LIN {X 0,Y 156.666,Z 359.376,A -85,B 0,C 180,E1 -23638.457,E2 -23638.457} C_VEL
LIN {X 0,Y 158.288,Z 353.415,A -85,B 0,C 180,E1 -23642.612,E2 -23642.612} C_VEL
LIN {X 0,Y 160.591,Z 345.69,A -85,B 0,C 180,E1 -23646.772,E2 -23646.772} C_VEL
LIN {X 0,Y 163.163,Z 336.899,A -85,B 0,C 180,E1 -23650.436,E2 -23650.436} C_VEL
LIN {X 0,Y 166.03,Z 327.188,A -85,B 0,C 180,E1 -23653.61,E2 -23653.61} C_VEL
LIN {X 0,Y 168.599,Z 317.53,A -85,B 0,C 180,E1 -23656.133,E2 -23656.133} C_VEL
LIN {X 0,Y 169.428,Z 313.24,A -85,B 0,C 180,E1 -23657.118,E2 -23657.118} C_VEL
LIN {X 0,Y 167.813,Z 301.872,A -85,B 0,C 180,E1 -23659.907,E2 -23659.907} C_VEL
LIN {X 0,Y 165.385,Z 290.388,A -85,B 0,C 180,E1 -23662.401,E2 -23662.401} C_VEL
LIN {X 0,Y 162.961,Z 281.712,A -85,B 0,C 180,E1 -23664.133,E2 -23664.133} C_VEL
LIN {X 0,Y 157.967,Z 269.688,A -85,B 0,C 180,E1 -23666.494,E2 -23666.494} C_VEL
LIN {X 0,Y 157.834,Z 268.828,A -85,B 0,C 180,E1 -23666.651,E2 -23666.651} C_VEL
LIN {X 0,Y 158.243,Z 268.777,A -85,B 0,C 180,E1 -23670.001,E2 -23670.001} C_VEL
LIN {X 0,Y 157.797,Z 268.827,A -85,B 0,C 180,E1 -23677.68,E2 -23677.68} C_VEL
LIN {X 0,Y 157.671,Z 268.84,A -85,B 0,C 180,E1 -23681.324,E2 -23681.324} C_VEL
LIN {X 0,Y 157.478,Z 268.873,A -85,B 0,C 180,E1 -23685.533,E2 -23685.533} C_VEL
LIN {X 0,Y 157.406,Z 268.881,A -85,B 0,C 180,E1 -23690.929,E2 -23690.929} C_VEL
LIN {X 0,Y 157.309,Z 268.883,A -85,B 0,C 180,E1 -23696.691,E2 -23696.691} C_VEL
LIN {X 0,Y 157.275,Z 268.897,A -85,B 0,C 180,E1 -23702.429,E2 -23702.429} C_VEL
LIN {X 0,Y 157.317,Z 268.876,A -85,B 0,C 180,E1 -23706.482,E2 -23706.482} C_VEL
LIN {X 0,Y 157.29,Z 268.893,A -85,B 0,C 180,E1 -23712.086,E2 -23712.086} C_VEL
LIN {X 0,Y 157.307,Z 268.881,A -85,B 0,C 180,E1 -23715.631,E2 -23715.631} C_VEL
LIN {X 0,Y 157.29,Z 268.889,A -85,B 0,C 180,E1 -23721.284,E2 -23721.284} C_VEL
LIN {X 0,Y 157.309,Z 268.889,A -85,B 0,C 180,E1 -23724.5,E2 -23724.5} C_VEL
LIN {X 0,Y 157.292,Z 268.878,A -85,B 0,C 180,E1 -23728.099,E2 -23728.099} C_VEL
LIN {X 0,Y 157.32,Z 268.883,A -85,B 0,C 180,E1 -23733.471,E2 -23733.471} C_VEL
LIN {X 0,Y 157.394,Z 268.872,A -85,B 0,C 180,E1 -23739.672,E2 -23739.672} C_VEL
LIN {X 0,Y 157.454,Z 268.858,A -85,B 0,C 180,E1 -23744.471,E2 -23744.471} C_VEL
LIN {X 0,Y 157.691,Z 268.843,A -85,B 0,C 180,E1 -23749.735,E2 -23749.735} C_VEL
LIN {X 0,Y 157.768,Z 268.826,A -85,B 0,C 180,E1 -23752.324,E2 -23752.324} C_VEL
LIN {X 0,Y 158.26,Z 268.771,A -85,B 0,C 180,E1 -23760.004,E2 -23760.004} C_VEL
LIN {X 0,Y 157.768,Z 268.819,A -85,B 0,C 180,E1 -23767.684,E2 -23767.684} C_VEL
LIN {X 0,Y 157.643,Z 268.848,A -85,B 0,C 180,E1 -23771.24,E2 -23771.24} C_VEL
LIN {X 0,Y 157.46,Z 268.861,A -85,B 0,C 180,E1 -23775.538,E2 -23775.538} C_VEL
LIN {X 0,Y 157.378,Z 268.881,A -85,B 0,C 180,E1 -23780.936,E2 -23780.936} C_VEL
LIN {X 0,Y 157.323,Z 268.889,A -85,B 0,C 180,E1 -23786.687,E2 -23786.687} C_VEL
LIN {X 0,Y 157.376,Z 269.021,A -85,B 0,C 180,E1 -23790.534,E2 -23790.534} C_VEL
LIN {X 0,Y 158.013,Z 272.957,A -85,B 0,C 180,E1 -23796.811,E2 -23796.811} C_VEL
LIN {X 0,Y 158.647,Z 276.209,A -85,B 0,C 180,E1 -23801.648,E2 -23801.648} C_VEL
LIN {X 0,Y 159.409,Z 279.832,A -85,B 0,C 180,E1 -23806.677,E2 -23806.677} C_VEL
LIN {X 0,Y 159.866,Z 282.353,A -85,B 0,C 180,E1 -23810.02,E2 -23810.02} C_VEL
LIN {X 0,Y 160.877,Z 285.754,A -85,B 0,C 180,E1 -23810.495,E2 -23810.495} C_VEL
LIN {X 0,Y 162.697,Z 294.146,A -85,B 0,C 180,E1 -23811.682,E2 -23811.682} C_VEL
LIN {X 0,Y 164.39,Z 306.903,A -85,B 0,C 180,E1 -23813.661,E2 -23813.661} C_VEL
LIN {X 0,Y 165.271,Z 319.319,A -85,B 0,C 180,E1 -23815.96,E2 -23815.96} C_VEL
LIN {X 0,Y 165.657,Z 331.535,A -85,B 0,C 180,E1 -23818.672,E2 -23818.672} C_VEL
LIN {X 0,Y 165.429,Z 342.008,A -85,B 0,C 180,E1 -23821.448,E2 -23821.448} C_VEL
LIN {X 0,Y 164.94,Z 346.369,A -85,B 0,C 180,E1 -23822.737,E2 -23822.737} C_VEL
LIN {X 0,Y 161.879,Z 356.685,A -85,B 0,C 180,E1 -23826.202,E2 -23826.202} C_VEL
LIN {X 0,Y 159.671,Z 364.153,A -85,B 0,C 180,E1 -23829.381,E2 -23829.381} C_VEL
LIN {X 0,Y 157.6,Z 371.203,A -85,B 0,C 180,E1 -23833.149,E2 -23833.149} C_VEL
LIN {X 0,Y 156.217,Z 376.821,A -85,B 0,C 180,E1 -23836.999,E2 -23836.999} C_VEL
LIN {X 0,Y 155.439,Z 381.221,A -85,B 0,C 180,E1 -23840.893,E2 -23840.893} C_VEL
LIN {X 0,Y 155.223,Z 384.632,A -85,B 0,C 180,E1 -23844.97,E2 -23844.97} C_VEL
LIN {X 0,Y 155.246,Z 386.125,A -85,B 0,C 180,E1 -23847.404,E2 -23847.404} C_VEL
LIN {X 0,Y 155.289,Z 387.302,A -85,B 0,C 180,E1 -23849.999,E2 -23849.999} C_VEL
LIN {X 0,Y 155.064,Z 388.289,A -85,B 0,C 180,E1 -23854.31,E2 -23854.31} C_VEL
LIN {X 0,Y 155.115,Z 388.283,A -85,B 0,C 180,E1 -23857.811,E2 -23857.811} C_VEL
LIN {X 0,Y 156.078,Z 387.02,A -85,B 0,C 180,E1 -23863.01,E2 -23863.01} C_VEL
LIN {X 0,Y 156.979,Z 385.836,A -85,B 0,C 180,E1 -23865.581,E2 -23865.581} C_VEL
LIN {X 0,Y 159.942,Z 382.247,A -85,B 0,C 180,E1 -23870.579,E2 -23870.579} C_VEL
LIN {X 0,Y 162.874,Z 378.482,A -85,B 0,C 180,E1 -23874.198,E2 -23874.198} C_VEL
LIN {X 0,Y 166.42,Z 373.702,A -85,B 0,C 180,E1 -23877.678,E2 -23877.678} C_VEL
LIN {X 0,Y 171.352,Z 366.713,A -85,B 0,C 180,E1 -23881.528,E2 -23881.528} C_VEL
LIN {X 0,Y 176.356,Z 359.27,A -85,B 0,C 180,E1 -23884.601,E2 -23884.601} C_VEL
LIN {X 0,Y 179.653,Z 351.998,A -85,B 0,C 180,E1 -23887.325,E2 -23887.325} C_VEL
LIN {X 0,Y 181.699,Z 345.766,A -85,B 0,C 180,E1 -23889.535,E2 -23889.535} C_VEL
LIN {X 0,Y 182.216,Z 342.101,A -85,B 0,C 180,E1 -23890.981,E2 -23890.981} C_VEL
LIN {X 0,Y 181.948,Z 338.759,A -85,B 0,C 180,E1 -23892.537,E2 -23892.537} C_VEL
LIN {X 0,Y 179.479,Z 328.783,A -85,B 0,C 180,E1 -23898.053,E2 -23898.053} C_VEL
LIN {X 0,Y 178.576,Z 323.642,A -85,B 0,C 180,E1 -23900.969,E2 -23900.969} C_VEL
LIN {X 0,Y 177.655,Z 319.569,A -85,B 0,C 180,E1 -23903.597,E2 -23903.597} C_VEL
LIN {X 0,Y 176.426,Z 314.669,A -85,B 0,C 180,E1 -23907.462,E2 -23907.462} C_VEL
LIN {X 0,Y 175.05,Z 309.179,A -85,B 0,C 180,E1 -23913.788,E2 -23913.788} C_VEL
LIN {X 0,Y 174.616,Z 307.537,A -85,B 0,C 180,E1 -23917.771,E2 -23917.771} C_VEL
LIN {X 0,Y 174.771,Z 306.887,A -85,B 0,C 180,E1 -23921.23,E2 -23921.23} C_VEL
LIN {X 0,Y 175.305,Z 306.933,A -85,B 0,C 180,E1 -23924.183,E2 -23924.183} C_VEL
LIN {X 0,Y 177.03,Z 310.07,A -85,B 0,C 180,E1 -23930.859,E2 -23930.859} C_VEL
LIN {X 0,Y 178.903,Z 314.102,A -85,B 0,C 180,E1 -23935.49,E2 -23935.49} C_VEL
LIN {X 0,Y 180.062,Z 318.511,A -85,B 0,C 180,E1 -23938.878,E2 -23938.878} C_VEL
LIN {X 0,Y 181.071,Z 323.62,A -85,B 0,C 180,E1 -23942.221,E2 -23942.221} C_VEL
LIN {X 0,Y 181.258,Z 328.749,A -85,B 0,C 180,E1 -23945.001,E2 -23945.001} C_VEL
LIN {X 0,Y 180.673,Z 334.595,A -85,B 0,C 180,E1 -23947.821,E2 -23947.821} C_VEL
LIN {X 0,Y 179.865,Z 337.31,A -85,B 0,C 180,E1 -23948.988,E2 -23948.988} C_VEL
LIN {X 0,Y 174.797,Z 345.135,A -85,B 0,C 180,E1 -23951.593,E2 -23951.593} C_VEL
LIN {X 0,Y 169.011,Z 352.991,A -85,B 0,C 180,E1 -23955.049,E2 -23955.049} C_VEL
LIN {X 0,Y 163.515,Z 359.573,A -85,B 0,C 180,E1 -23958.994,E2 -23958.994} C_VEL
LIN {X 0,Y 159.609,Z 363.69,A -85,B 0,C 180,E1 -23962.384,E2 -23962.384} C_VEL
LIN {X 0,Y 155.548,Z 367.521,A -85,B 0,C 180,E1 -23966.855,E2 -23966.855} C_VEL
LIN {X 0,Y 153.024,Z 369.486,A -85,B 0,C 180,E1 -23970.339,E2 -23970.339} C_VEL
LIN {X 0,Y 150.989,Z 370.683,A -85,B 0,C 180,E1 -23973.95,E2 -23973.95} C_VEL
LIN {X 0,Y 149.468,Z 371.159,A -85,B 0,C 180,E1 -23977.674,E2 -23977.674} C_VEL
LIN {X 0,Y 148.38,Z 370.887,A -85,B 0,C 180,E1 -23981.53,E2 -23981.53} C_VEL
LIN {X 0,Y 147.801,Z 369.765,A -85,B 0,C 180,E1 -23985.493,E2 -23985.493} C_VEL
LIN {X 0,Y 147.748,Z 367.741,A -85,B 0,C 180,E1 -23989.552,E2 -23989.552} C_VEL
LIN {X 0,Y 148.32,Z 364.749,A -85,B 0,C 180,E1 -23993.652,E2 -23993.652} C_VEL
LIN {X 0,Y 149.366,Z 360.568,A -85,B 0,C 180,E1 -23997.87,E2 -23997.87} C_VEL
LIN {X 0,Y 150.925,Z 354.855,A -85,B 0,C 180,E1 -24002.249,E2 -24002.249} C_VEL
LIN {X 0,Y 153.216,Z 347.505,A -85,B 0,C 180,E1 -24006.535,E2 -24006.535} C_VEL
LIN {X 0,Y 155.853,Z 338.829,A -85,B 0,C 180,E1 -24010.487,E2 -24010.487} C_VEL
LIN {X 0,Y 158.843,Z 328.979,A -85,B 0,C 180,E1 -24013.948,E2 -24013.948} C_VEL
LIN {X 0,Y 161.788,Z 318.591,A -85,B 0,C 180,E1 -24016.819,E2 -24016.819} C_VEL
LIN {X 0,Y 162.665,Z 314.349,A -85,B 0,C 180,E1 -24017.842,E2 -24017.842} C_VEL
LIN {X 0,Y 161.407,Z 304.628,A -85,B 0,C 180,E1 -24020.395,E2 -24020.395} C_VEL
LIN {X 0,Y 159.163,Z 293.185,A -85,B 0,C 180,E1 -24023.068,E2 -24023.068} C_VEL
LIN {X 0,Y 156.904,Z 284.815,A -85,B 0,C 180,E1 -24024.862,E2 -24024.862} C_VEL
LIN {X 0,Y 151.838,Z 272.437,A -85,B 0,C 180,E1 -24027.556,E2 -24027.556} C_VEL
LIN {X 0,Y 150.939,Z 269.688,A -85,B 0,C 180,E1 -24028.084,E2 -24028.084} C_VEL
LIN {X 0,Y 151.203,Z 269.654,A -85,B 0,C 180,E1 -24030.001,E2 -24030.001} C_VEL
LIN {X 0,Y 150.732,Z 269.709,A -85,B 0,C 180,E1 -24038.042,E2 -24038.042} C_VEL
LIN {X 0,Y 150.602,Z 269.72,A -85,B 0,C 180,E1 -24041.51,E2 -24041.51} C_VEL
LIN {X 0,Y 150.387,Z 269.757,A -85,B 0,C 180,E1 -24046.285,E2 -24046.285} C_VEL
LIN {X 0,Y 150.379,Z 269.756,A -85,B 0,C 180,E1 -24050.835,E2 -24050.835} C_VEL
LIN {X 0,Y 150.238,Z 269.763,A -85,B 0,C 180,E1 -24057.288,E2 -24057.288} C_VEL
LIN {X 0,Y 150.215,Z 269.775,A -85,B 0,C 180,E1 -24062.641,E2 -24062.641} C_VEL
LIN {X 0,Y 150.229,Z 269.761,A -85,B 0,C 180,E1 -24067.459,E2 -24067.459} C_VEL
LIN {X 0,Y 150.231,Z 269.771,A -85,B 0,C 180,E1 -24071.547,E2 -24071.547} C_VEL
LIN {X 0,Y 150.282,Z 269.756,A -85,B 0,C 180,E1 -24075.461,E2 -24075.461} C_VEL
LIN {X 0,Y 150.232,Z 269.759,A -85,B 0,C 180,E1 -24079.092,E2 -24079.092} C_VEL
LIN {X 0,Y 150.268,Z 269.767,A -85,B 0,C 180,E1 -24082.665,E2 -24082.665} C_VEL
LIN {X 0,Y 150.218,Z 269.764,A -85,B 0,C 180,E1 -24087.369,E2 -24087.369} C_VEL
LIN {X 0,Y 150.242,Z 269.762,A -85,B 0,C 180,E1 -24092.723,E2 -24092.723} C_VEL
LIN {X 0,Y 150.35,Z 269.751,A -85,B 0,C 180,E1 -24099.213,E2 -24099.213} C_VEL
LIN {X 0,Y 150.361,Z 269.736,A -85,B 0,C 180,E1 -24103.718,E2 -24103.718} C_VEL
LIN {X 0,Y 150.613,Z 269.723,A -85,B 0,C 180,E1 -24109.247,E2 -24109.247} C_VEL
LIN {X 0,Y 150.706,Z 269.707,A -85,B 0,C 180,E1 -24111.962,E2 -24111.962} C_VEL
LIN {X 0,Y 151.221,Z 269.648,A -85,B 0,C 180,E1 -24120.004,E2 -24120.004} C_VEL
LIN {X 0,Y 150.706,Z 269.701,A -85,B 0,C 180,E1 -24128.047,E2 -24128.047} C_VEL
LIN {X 0,Y 150.583,Z 269.728,A -85,B 0,C 180,E1 -24131.44,E2 -24131.44} C_VEL
LIN {X 0,Y 150.367,Z 269.743,A -85,B 0,C 180,E1 -24136.29,E2 -24136.29} C_VEL
LIN {X 0,Y 150.359,Z 269.755,A -85,B 0,C 180,E1 -24140.796,E2 -24140.796} C_VEL
LIN {X 0,Y 150.254,Z 269.769,A -85,B 0,C 180,E1 -24147.286,E2 -24147.286} C_VEL
LIN {X 0,Y 150.284,Z 269.815,A -85,B 0,C 180,E1 -24149.798,E2 -24149.798} C_VEL
LIN {X 0,Y 150.664,Z 272.327,A -85,B 0,C 180,E1 -24154.044,E2 -24154.044} C_VEL
LIN {X 0,Y 151.126,Z 274.608,A -85,B 0,C 180,E1 -24157.759,E2 -24157.759} C_VEL
LIN {X 0,Y 151.921,Z 278.719,A -85,B 0,C 180,E1 -24163.946,E2 -24163.946} C_VEL
LIN {X 0,Y 152.638,Z 282.108,A -85,B 0,C 180,E1 -24168.532,E2 -24168.532} C_VEL
LIN {X 0,Y 153.768,Z 285.468,A -85,B 0,C 180,E1 -24169.066,E2 -24169.066} C_VEL
LIN {X 0,Y 155.923,Z 293.086,A -85,B 0,C 180,E1 -24170.301,E2 -24170.301} C_VEL
LIN {X 0,Y 157.671,Z 305.728,A -85,B 0,C 180,E1 -24172.338,E2 -24172.338} C_VEL
LIN {X 0,Y 158.46,Z 316.907,A -85,B 0,C 180,E1 -24174.449,E2 -24174.449} C_VEL
LIN {X 0,Y 158.758,Z 329.337,A -85,B 0,C 180,E1 -24177.263,E2 -24177.263} C_VEL
LIN {X 0,Y 158.629,Z 339.851,A -85,B 0,C 180,E1 -24180.103,E2 -24180.103} C_VEL
LIN {X 0,Y 158.315,Z 345.557,A -85,B 0,C 180,E1 -24181.856,E2 -24181.856} C_VEL
LIN {X 0,Y 155.24,Z 355.549,A -85,B 0,C 180,E1 -24185.303,E2 -24185.303} C_VEL
LIN {X 0,Y 152.604,Z 364.128,A -85,B 0,C 180,E1 -24189.088,E2 -24189.088} C_VEL
LIN {X 0,Y 150.499,Z 371.077,A -85,B 0,C 180,E1 -24193.029,E2 -24193.029} C_VEL
LIN {X 0,Y 148.93,Z 377.433,A -85,B 0,C 180,E1 -24197.738,E2 -24197.738} C_VEL
LIN {X 0,Y 148.275,Z 381.585,A -85,B 0,C 180,E1 -24201.824,E2 -24201.824} C_VEL
LIN {X 0,Y 148.144,Z 384.111,A -85,B 0,C 180,E1 -24205.077,E2 -24205.077} C_VEL
LIN {X 0,Y 148.167,Z 385.441,A -85,B 0,C 180,E1 -24207.28,E2 -24207.28} C_VEL
LIN {X 0,Y 148.227,Z 386.676,A -85,B 0,C 180,E1 -24209.999,E2 -24209.999} C_VEL
LIN {X 0,Y 148.002,Z 387.734,A -85,B 0,C 180,E1 -24214.235,E2 -24214.235} C_VEL
LIN {X 0,Y 148.051,Z 387.874,A -85,B 0,C 180,E1 -24218.186,E2 -24218.186} C_VEL
LIN {X 0,Y 149.126,Z 386.732,A -85,B 0,C 180,E1 -24223.628,E2 -24223.628} C_VEL
LIN {X 0,Y 151.54,Z 384.125,A -85,B 0,C 180,E1 -24228.942,E2 -24228.942} C_VEL
LIN {X 0,Y 155.254,Z 379.899,A -85,B 0,C 180,E1 -24234.041,E2 -24234.041} C_VEL
LIN {X 0,Y 159.192,Z 375.209,A -85,B 0,C 180,E1 -24237.991,E2 -24237.991} C_VEL
LIN {X 0,Y 164.552,Z 368.297,A -85,B 0,C 180,E1 -24242.266,E2 -24242.266} C_VEL
LIN {X 0,Y 169.739,Z 361.27,A -85,B 0,C 180,E1 -24245.425,E2 -24245.425} C_VEL
LIN {X 0,Y 172.726,Z 355.886,A -85,B 0,C 180,E1 -24247.612,E2 -24247.612} C_VEL
LIN {X 0,Y 175.271,Z 349.958,A -85,B 0,C 180,E1 -24249.907,E2 -24249.907} C_VEL
LIN {X 0,Y 177.96,Z 341.077,A -85,B 0,C 180,E1 -24253.174,E2 -24253.174} C_VEL
LIN {X 0,Y 179.367,Z 333.898,A -85,B 0,C 180,E1 -24255.826,E2 -24255.826} C_VEL
LIN {X 0,Y 179.683,Z 330.758,A -85,B 0,C 180,E1 -24257.067,E2 -24257.067} C_VEL
LIN {X 0,Y 179.479,Z 328.783,A -85,B 0,C 180,E1 -24258.053,E2 -24258.053} C_VEL
LIN {X 0,Y 178.99,Z 326.998,A -85,B 0,C 180,E1 -24259.16,E2 -24259.16} C_VEL
LIN {X 0,Y 178.139,Z 325.698,A -85,B 0,C 180,E1 -24260.321,E2 -24260.321} C_VEL
LIN {X 0,Y 175.905,Z 324.041,A -85,B 0,C 180,E1 -24262.735,E2 -24262.735} C_VEL
LIN {X 0,Y 172.932,Z 321.835,A -85,B 0,C 180,E1 -24266.535,E2 -24266.535} C_VEL
LIN {X 0,Y 172.514,Z 320.598,A -85,B 0,C 180,E1 -24267.798,E2 -24267.798} C_VEL
LIN {X 0,Y 171.551,Z 315.189,A -85,B 0,C 180,E1 -24274.323,E2 -24274.323} C_VEL
LIN {X 0,Y 171.295,Z 313.685,A -85,B 0,C 180,E1 -24278.326,E2 -24278.326} C_VEL
LIN {X 0,Y 171.793,Z 313.062,A -85,B 0,C 180,E1 -24283.356,E2 -24283.356} C_VEL
LIN {X 0,Y 173.242,Z 316.068,A -85,B 0,C 180,E1 -24290.657,E2 -24290.657} C_VEL
LIN {X 0,Y 174.721,Z 319.97,A -85,B 0,C 180,E1 -24295.382,E2 -24295.382} C_VEL
LIN {X 0,Y 175.516,Z 324.272,A -85,B 0,C 180,E1 -24298.85,E2 -24298.85} C_VEL
LIN {X 0,Y 175.951,Z 327.513,A -85,B 0,C 180,E1 -24301.141,E2 -24301.141} C_VEL
LIN {X 0,Y 175.903,Z 332.178,A -85,B 0,C 180,E1 -24303.947,E2 -24303.947} C_VEL
LIN {X 0,Y 175.004,Z 337.799,A -85,B 0,C 180,E1 -24306.916,E2 -24306.916} C_VEL
LIN {X 0,Y 174.65,Z 338.985,A -85,B 0,C 180,E1 -24307.479,E2 -24307.479} C_VEL
LIN {X 0,Y 169.371,Z 346.589,A -85,B 0,C 180,E1 -24310.153,E2 -24310.153} C_VEL
LIN {X 0,Y 163.267,Z 354.247,A -85,B 0,C 180,E1 -24313.689,E2 -24313.689} C_VEL
LIN {X 0,Y 157.729,Z 360.377,A -85,B 0,C 180,E1 -24317.524,E2 -24317.524} C_VEL
LIN {X 0,Y 152.999,Z 364.947,A -85,B 0,C 180,E1 -24321.555,E2 -24321.555} C_VEL
LIN {X 0,Y 148.757,Z 368.47,A -85,B 0,C 180,E1 -24326.153,E2 -24326.153} C_VEL
LIN {X 0,Y 146.004,Z 370.323,A -85,B 0,C 180,E1 -24329.956,E2 -24329.956} C_VEL
LIN {X 0,Y 143.85,Z 371.381,A -85,B 0,C 180,E1 -24333.847,E2 -24333.847} C_VEL
LIN {X 0,Y 142.294,Z 371.629,A -85,B 0,C 180,E1 -24337.794,E2 -24337.794} C_VEL
LIN {X 0,Y 141.22,Z 371.128,A -85,B 0,C 180,E1 -24341.715,E2 -24341.715} C_VEL
LIN {X 0,Y 140.69,Z 369.923,A -85,B 0,C 180,E1 -24345.627,E2 -24345.627} C_VEL
LIN {X 0,Y 140.812,Z 366.84,A -85,B 0,C 180,E1 -24351.28,E2 -24351.28} C_VEL
LIN {X 0,Y 141.526,Z 363.716,A -85,B 0,C 180,E1 -24355.177,E2 -24355.177} C_VEL
LIN {X 0,Y 142.807,Z 358.87,A -85,B 0,C 180,E1 -24359.755,E2 -24359.755} C_VEL
LIN {X 0,Y 144.887,Z 351.955,A -85,B 0,C 180,E1 -24364.675,E2 -24364.675} C_VEL
LIN {X 0,Y 147.505,Z 343.824,A -85,B 0,C 180,E1 -24369.065,E2 -24369.065} C_VEL
LIN {X 0,Y 150.561,Z 334.302,A -85,B 0,C 180,E1 -24373.039,E2 -24373.039} C_VEL
LIN {X 0,Y 153.777,Z 323.765,A -85,B 0,C 180,E1 -24376.435,E2 -24376.435} C_VEL
LIN {X 0,Y 155.921,Z 315.38,A -85,B 0,C 180,E1 -24378.628,E2 -24378.628} C_VEL
LIN {X 0,Y 154.571,Z 304.968,A -85,B 0,C 180,E1 -24381.504,E2 -24381.504} C_VEL
LIN {X 0,Y 152.387,Z 293.541,A -85,B 0,C 180,E1 -24384.316,E2 -24384.316} C_VEL
LIN {X 0,Y 150.185,Z 286.052,A -85,B 0,C 180,E1 -24386.076,E2 -24386.076} C_VEL
LIN {X 0,Y 145.1,Z 273.536,A -85,B 0,C 180,E1 -24389,E2 -24389} C_VEL
LIN {X 0,Y 144.09,Z 270.538,A -85,B 0,C 180,E1 -24389.617,E2 -24389.617} C_VEL
LIN {X 0,Y 143.608,Z 270.594,A -85,B 0,C 180,E1 -24395.618,E2 -24395.618} C_VEL
LIN {X 0,Y 143.653,Z 270.591,A -85,B 0,C 180,E1 -24398.441,E2 -24398.441} C_VEL
LIN {X 0,Y 143.536,Z 270.6,A -85,B 0,C 180,E1 -24401.715,E2 -24401.715} C_VEL
LIN {X 0,Y 143.325,Z 270.632,A -85,B 0,C 180,E1 -24407.112,E2 -24407.112} C_VEL
LIN {X 0,Y 143.301,Z 270.64,A -85,B 0,C 180,E1 -24411.293,E2 -24411.293} C_VEL
LIN {X 0,Y 143.184,Z 270.644,A -85,B 0,C 180,E1 -24417.944,E2 -24417.944} C_VEL
LIN {X 0,Y 143.164,Z 270.65,A -85,B 0,C 180,E1 -24423.442,E2 -24423.442} C_VEL
LIN {X 0,Y 143.123,Z 270.654,A -85,B 0,C 180,E1 -24429.671,E2 -24429.671} C_VEL
LIN {X 0,Y 143.176,Z 270.648,A -85,B 0,C 180,E1 -24433.411,E2 -24433.411} C_VEL
LIN {X 0,Y 143.165,Z 270.631,A -85,B 0,C 180,E1 -24437.424,E2 -24437.424} C_VEL
LIN {X 0,Y 143.185,Z 270.646,A -85,B 0,C 180,E1 -24441.754,E2 -24441.754} C_VEL
LIN {X 0,Y 143.186,Z 270.64,A -85,B 0,C 180,E1 -24447.328,E2 -24447.328} C_VEL
LIN {X 0,Y 143.188,Z 270.636,A -85,B 0,C 180,E1 -24452.068,E2 -24452.068} C_VEL
LIN {X 0,Y 143.276,Z 270.632,A -85,B 0,C 180,E1 -24458.751,E2 -24458.751} C_VEL
LIN {X 0,Y 143.301,Z 270.612,A -85,B 0,C 180,E1 -24462.892,E2 -24462.892} C_VEL
LIN {X 0,Y 143.539,Z 270.604,A -85,B 0,C 180,E1 -24468.711,E2 -24468.711} C_VEL
LIN {X 0,Y 143.627,Z 270.591,A -85,B 0,C 180,E1 -24471.564,E2 -24471.564} C_VEL
LIN {X 0,Y 144.179,Z 270.525,A -85,B 0,C 180,E1 -24480.005,E2 -24480.005} C_VEL
LIN {X 0,Y 143.628,Z 270.585,A -85,B 0,C 180,E1 -24488.446,E2 -24488.446} C_VEL
LIN {X 0,Y 143.511,Z 270.61,A -85,B 0,C 180,E1 -24491.633,E2 -24491.633} C_VEL
LIN {X 0,Y 143.307,Z 270.624,A -85,B 0,C 180,E1 -24497.117,E2 -24497.117} C_VEL
LIN {X 0,Y 143.285,Z 270.637,A -85,B 0,C 180,E1 -24501.258,E2 -24501.258} C_VEL
LIN {X 0,Y 143.19,Z 270.649,A -85,B 0,C 180,E1 -24508.528,E2 -24508.528} C_VEL
LIN {X 0,Y 143.259,Z 270.819,A -85,B 0,C 180,E1 -24509.384,E2 -24509.384} C_VEL
LIN {X 0,Y 143.624,Z 273.231,A -85,B 0,C 180,E1 -24513.707,E2 -24513.707} C_VEL
LIN {X 0,Y 144.229,Z 276.602,A -85,B 0,C 180,E1 -24519.312,E2 -24519.312} C_VEL
LIN {X 0,Y 144.985,Z 280.082,A -85,B 0,C 180,E1 -24524.759,E2 -24524.759} C_VEL
LIN {X 0,Y 145.303,Z 281.422,A -85,B 0,C 180,E1 -24526.772,E2 -24526.772} C_VEL
LIN {X 0,Y 146.379,Z 284.855,A -85,B 0,C 180,E1 -24527.377,E2 -24527.377} C_VEL
LIN {X 0,Y 148.888,Z 291.712,A -85,B 0,C 180,E1 -24528.701,E2 -24528.701} C_VEL
LIN {X 0,Y 150.419,Z 300.402,A -85,B 0,C 180,E1 -24530.181,E2 -24530.181} C_VEL
LIN {X 0,Y 151.509,Z 312.008,A -85,B 0,C 180,E1 -24532.356,E2 -24532.356} C_VEL
LIN {X 0,Y 151.963,Z 324.4,A -85,B 0,C 180,E1 -24535.086,E2 -24535.086} C_VEL
LIN {X 0,Y 151.991,Z 335.023,A -85,B 0,C 180,E1 -24537.874,E2 -24537.874} C_VEL
LIN {X 0,Y 151.536,Z 344.673,A -85,B 0,C 180,E1 -24540.857,E2 -24540.857} C_VEL
LIN {X 0,Y 149.617,Z 351.472,A -85,B 0,C 180,E1 -24543.197,E2 -24543.197} C_VEL
LIN {X 0,Y 146.829,Z 360.018,A -85,B 0,C 180,E1 -24546.739,E2 -24546.739} C_VEL
LIN {X 0,Y 144.387,Z 367.699,A -85,B 0,C 180,E1 -24550.817,E2 -24550.817} C_VEL
LIN {X 0,Y 142.365,Z 374.736,A -85,B 0,C 180,E1 -24555.708,E2 -24555.708} C_VEL
LIN {X 0,Y 141.428,Z 379.41,A -85,B 0,C 180,E1 -24559.982,E2 -24559.982} C_VEL
LIN {X 0,Y 141.09,Z 383.499,A -85,B 0,C 180,E1 -24565.077,E2 -24565.077} C_VEL
LIN {X 0,Y 141.165,Z 386.031,A -85,B 0,C 180,E1 -24569.998,E2 -24569.998} C_VEL
LIN {X 0,Y 140.938,Z 387.167,A -85,B 0,C 180,E1 -24574.145,E2 -24574.145} C_VEL
LIN {X 0,Y 141.012,Z 387.435,A -85,B 0,C 180,E1 -24578.597,E2 -24578.597} C_VEL
LIN {X 0,Y 142.203,Z 386.446,A -85,B 0,C 180,E1 -24584.305,E2 -24584.305} C_VEL
LIN {X 0,Y 144.81,Z 383.984,A -85,B 0,C 180,E1 -24589.859,E2 -24589.859} C_VEL
LIN {X 0,Y 147.67,Z 381.121,A -85,B 0,C 180,E1 -24593.86,E2 -24593.86} C_VEL
LIN {X 0,Y 151.293,Z 377.328,A -85,B 0,C 180,E1 -24597.678,E2 -24597.678} C_VEL
LIN {X 0,Y 155.418,Z 372.527,A -85,B 0,C 180,E1 -24601.332,E2 -24601.332} C_VEL
LIN {X 0,Y 161.229,Z 365.531,A -85,B 0,C 180,E1 -24605.278,E2 -24605.278} C_VEL
LIN {X 0,Y 164.903,Z 360.739,A -85,B 0,C 180,E1 -24607.394,E2 -24607.394} C_VEL
LIN {X 0,Y 168.575,Z 354.012,A -85,B 0,C 180,E1 -24610.254,E2 -24610.254} C_VEL
LIN {X 0,Y 171.589,Z 346.4,A -85,B 0,C 180,E1 -24613.316,E2 -24613.316} C_VEL
LIN {X 0,Y 173.669,Z 339.3,A -85,B 0,C 180,E1 -24616.107,E2 -24616.107} C_VEL
LIN {X 0,Y 174.513,Z 334.939,A -85,B 0,C 180,E1 -24617.894,E2 -24617.894} C_VEL
LIN {X 0,Y 174.264,Z 331.227,A -85,B 0,C 180,E1 -24620.017,E2 -24620.017} C_VEL
LIN {X 0,Y 173.354,Z 324.946,A -85,B 0,C 180,E1 -24624.174,E2 -24624.174} C_VEL
LIN {X 0,Y 172.514,Z 320.598,A -85,B 0,C 180,E1 -24627.798,E2 -24627.798} C_VEL
LIN {X 0,Y 172.161,Z 319.51,A -85,B 0,C 180,E1 -24629.045,E2 -24629.045} C_VEL
LIN {X 0,Y 171.528,Z 318.985,A -85,B 0,C 180,E1 -24630.327,E2 -24630.327} C_VEL
LIN {X 0,Y 169.874,Z 319.056,A -85,B 0,C 180,E1 -24632.935,E2 -24632.935} C_VEL
LIN {X 0,Y 167.791,Z 319.912,A -85,B 0,C 180,E1 -24637.003,E2 -24637.003} C_VEL
LIN {X 0,Y 167.583,Z 319.815,A -85,B 0,C 180,E1 -24638.385,E2 -24638.385} C_VEL
LIN {X 0,Y 168.009,Z 319.159,A -85,B 0,C 180,E1 -24642.969,E2 -24642.969} C_VEL
LIN {X 0,Y 168.514,Z 320.844,A -85,B 0,C 180,E1 -24647.96,E2 -24647.96} C_VEL
LIN {X 0,Y 169.162,Z 321.867,A -85,B 0,C 180,E1 -24650.43,E2 -24650.43} C_VEL
LIN {X 0,Y 170.272,Z 325.619,A -85,B 0,C 180,E1 -24655.261,E2 -24655.261} C_VEL
LIN {X 0,Y 170.688,Z 329.788,A -85,B 0,C 180,E1 -24658.816,E2 -24658.816} C_VEL
LIN {X 0,Y 170.745,Z 332.98,A -85,B 0,C 180,E1 -24661.175,E2 -24661.175} C_VEL
LIN {X 0,Y 170.376,Z 336.631,A -85,B 0,C 180,E1 -24663.491,E2 -24663.491} C_VEL
LIN {X 0,Y 169.489,Z 340.363,A -85,B 0,C 180,E1 -24665.643,E2 -24665.643} C_VEL
LIN {X 0,Y 168.571,Z 342.144,A -85,B 0,C 180,E1 -24666.427,E2 -24666.427} C_VEL
LIN {X 0,Y 162.772,Z 349.69,A -85,B 0,C 180,E1 -24669.307,E2 -24669.307} C_VEL
LIN {X 0,Y 156.423,Z 356.83,A -85,B 0,C 180,E1 -24672.978,E2 -24672.978} C_VEL
LIN {X 0,Y 151.821,Z 361.41,A -85,B 0,C 180,E1 -24676.121,E2 -24676.121} C_VEL
LIN {X 0,Y 146.052,Z 366.443,A -85,B 0,C 180,E1 -24680.96,E2 -24680.96} C_VEL
LIN {X 0,Y 141.199,Z 369.919,A -85,B 0,C 180,E1 -24686.376,E2 -24686.376} C_VEL
LIN {X 0,Y 138.403,Z 371.42,A -85,B 0,C 180,E1 -24690.511,E2 -24690.511} C_VEL
LIN {X 0,Y 136.351,Z 372.066,A -85,B 0,C 180,E1 -24694.533,E2 -24694.533} C_VEL
LIN {X 0,Y 134.87,Z 371.937,A -85,B 0,C 180,E1 -24698.698,E2 -24698.698} C_VEL
LIN {X 0,Y 133.881,Z 371.03,A -85,B 0,C 180,E1 -24703.026,E2 -24703.026} C_VEL
LIN {X 0,Y 133.516,Z 369.271,A -85,B 0,C 180,E1 -24707.462,E2 -24707.462} C_VEL
LIN {X 0,Y 134.056,Z 365.488,A -85,B 0,C 180,E1 -24713.432,E2 -24713.432} C_VEL
LIN {X 0,Y 135.338,Z 360.61,A -85,B 0,C 180,E1 -24718.717,E2 -24718.717} C_VEL
LIN {X 0,Y 137.015,Z 354.909,A -85,B 0,C 180,E1 -24723.334,E2 -24723.334} C_VEL
LIN {X 0,Y 139.426,Z 347.744,A -85,B 0,C 180,E1 -24727.817,E2 -24727.817} C_VEL
LIN {X 0,Y 141.784,Z 340.585,A -85,B 0,C 180,E1 -24731.38,E2 -24731.38} C_VEL
LIN {X 0,Y 144.774,Z 331.627,A -85,B 0,C 180,E1 -24734.945,E2 -24734.945} C_VEL
LIN {X 0,Y 147.769,Z 321.914,A -85,B 0,C 180,E1 -24737.992,E2 -24737.992} C_VEL
LIN {X 0,Y 149.163,Z 316.352,A -85,B 0,C 180,E1 -24739.482,E2 -24739.482} C_VEL
LIN {X 0,Y 147.887,Z 306.104,A -85,B 0,C 180,E1 -24742.492,E2 -24742.492} C_VEL
LIN {X 0,Y 146.074,Z 295.928,A -85,B 0,C 180,E1 -24745.172,E2 -24745.172} C_VEL
LIN {X 0,Y 144.175,Z 289.226,A -85,B 0,C 180,E1 -24746.884,E2 -24746.884} C_VEL
LIN {X 0,Y 139.016,Z 276.237,A -85,B 0,C 180,E1 -24750.183,E2 -24750.183} C_VEL
LIN {X 0,Y 137.798,Z 273.934,A -85,B 0,C 180,E1 -24750.824,E2 -24750.824} C_VEL
LIN {X 0,Y 136.906,Z 271.433,A -85,B 0,C 180,E1 -24751.472,E2 -24751.472} C_VEL
LIN {X 0,Y 136.58,Z 271.473,A -85,B 0,C 180,E1 -24758.882,E2 -24758.882} C_VEL
LIN {X 0,Y 136.479,Z 271.478,A -85,B 0,C 180,E1 -24761.957,E2 -24761.957} C_VEL
LIN {X 0,Y 136.264,Z 271.508,A -85,B 0,C 180,E1 -24768.028,E2 -24768.028} C_VEL
LIN {X 0,Y 136.217,Z 271.523,A -85,B 0,C 180,E1 -24771.784,E2 -24771.784} C_VEL
LIN {X 0,Y 136.11,Z 271.527,A -85,B 0,C 180,E1 -24778.635,E2 -24778.635} C_VEL
LIN {X 0,Y 136.076,Z 271.526,A -85,B 0,C 180,E1 -24784.621,E2 -24784.621} C_VEL
LIN {X 0,Y 136.097,Z 271.529,A -85,B 0,C 180,E1 -24789.241,E2 -24789.241} C_VEL
LIN {X 0,Y 136.111,Z 271.528,A -85,B 0,C 180,E1 -24793.715,E2 -24793.715} C_VEL
LIN {X 0,Y 136.113,Z 271.509,A -85,B 0,C 180,E1 -24797.845,E2 -24797.845} C_VEL
LIN {X 0,Y 136.136,Z 271.524,A -85,B 0,C 180,E1 -24801.728,E2 -24801.728} C_VEL
LIN {X 0,Y 136.095,Z 271.53,A -85,B 0,C 180,E1 -24805.718,E2 -24805.718} C_VEL
LIN {X 0,Y 136.144,Z 271.514,A -85,B 0,C 180,E1 -24812.322,E2 -24812.322} C_VEL
LIN {X 0,Y 136.243,Z 271.508,A -85,B 0,C 180,E1 -24818.839,E2 -24818.839} C_VEL
LIN {X 0,Y 136.269,Z 271.499,A -85,B 0,C 180,E1 -24825.061,E2 -24825.061} C_VEL
LIN {X 0,Y 136.446,Z 271.489,A -85,B 0,C 180,E1 -24828.143,E2 -24828.143} C_VEL
LIN {X 0,Y 136.553,Z 271.473,A -85,B 0,C 180,E1 -24831.123,E2 -24831.123} C_VEL
LIN {X 0,Y 137.136,Z 271.402,A -85,B 0,C 180,E1 -24840.005,E2 -24840.005} C_VEL
LIN {X 0,Y 136.554,Z 271.468,A -85,B 0,C 180,E1 -24848.887,E2 -24848.887} C_VEL
LIN {X 0,Y 136.447,Z 271.489,A -85,B 0,C 180,E1 -24851.895,E2 -24851.895} C_VEL
LIN {X 0,Y 136.249,Z 271.508,A -85,B 0,C 180,E1 -24858.034,E2 -24858.034} C_VEL
LIN {X 0,Y 136.206,Z 271.519,A -85,B 0,C 180,E1 -24861.753,E2 -24861.753} C_VEL
LIN {X 0,Y 136.167,Z 271.648,A -85,B 0,C 180,E1 -24868.664,E2 -24868.664} C_VEL
LIN {X 0,Y 136.664,Z 274.855,A -85,B 0,C 180,E1 -24874.631,E2 -24874.631} C_VEL
LIN {X 0,Y 137.244,Z 277.852,A -85,B 0,C 180,E1 -24879.812,E2 -24879.812} C_VEL
LIN {X 0,Y 137.974,Z 280.975,A -85,B 0,C 180,E1 -24884.913,E2 -24884.913} C_VEL
LIN {X 0,Y 139.029,Z 284.358,A -85,B 0,C 180,E1 -24885.569,E2 -24885.569} C_VEL
LIN {X 0,Y 142.365,Z 292.858,A -85,B 0,C 180,E1 -24887.386,E2 -24887.386} C_VEL
LIN {X 0,Y 143.74,Z 299.24,A -85,B 0,C 180,E1 -24888.603,E2 -24888.603} C_VEL
LIN {X 0,Y 144.863,Z 311.03,A -85,B 0,C 180,E1 -24890.924,E2 -24890.924} C_VEL
LIN {X 0,Y 145.22,Z 322.971,A -85,B 0,C 180,E1 -24893.661,E2 -24893.661} C_VEL
LIN {X 0,Y 145.182,Z 334.443,A -85,B 0,C 180,E1 -24896.797,E2 -24896.797} C_VEL
LIN {X 0,Y 144.645,Z 344.71,A -85,B 0,C 180,E1 -24900.129,E2 -24900.129} C_VEL
LIN {X 0,Y 142.366,Z 352.386,A -85,B 0,C 180,E1 -24902.936,E2 -24902.936} C_VEL
LIN {X 0,Y 139.36,Z 361.283,A -85,B 0,C 180,E1 -24906.992,E2 -24906.992} C_VEL
LIN {X 0,Y 136.952,Z 368.622,A -85,B 0,C 180,E1 -24911.291,E2 -24911.291} C_VEL
LIN {X 0,Y 135.064,Z 375.368,A -85,B 0,C 180,E1 -24916.457,E2 -24916.457} C_VEL
LIN {X 0,Y 134.232,Z 379.79,A -85,B 0,C 180,E1 -24920.961,E2 -24920.961} C_VEL
LIN {X 0,Y 134.037,Z 382.851,A -85,B 0,C 180,E1 -24925.071,E2 -24925.071} C_VEL
LIN {X 0,Y 134.103,Z 385.377,A -85,B 0,C 180,E1 -24929.998,E2 -24929.998} C_VEL
LIN {X 0,Y 133.866,Z 386.506,A -85,B 0,C 180,E1 -24933.991,E2 -24933.991} C_VEL
LIN {X 0,Y 133.993,Z 386.966,A -85,B 0,C 180,E1 -24939.051,E2 -24939.051} C_VEL
LIN {X 0,Y 135.309,Z 386.17,A -85,B 0,C 180,E1 -24945.051,E2 -24945.051} C_VEL
LIN {X 0,Y 138.124,Z 383.851,A -85,B 0,C 180,E1 -24950.864,E2 -24950.864} C_VEL
LIN {X 0,Y 142.396,Z 380.03,A -85,B 0,C 180,E1 -24956.37,E2 -24956.37} C_VEL
LIN {X 0,Y 146.136,Z 376.343,A -85,B 0,C 180,E1 -24960.034,E2 -24960.034} C_VEL
LIN {X 0,Y 151.026,Z 371.122,A -85,B 0,C 180,E1 -24963.945,E2 -24963.945} C_VEL
LIN {X 0,Y 157.46,Z 363.877,A -85,B 0,C 180,E1 -24967.856,E2 -24967.856} C_VEL
LIN {X 0,Y 160.134,Z 360.242,A -85,B 0,C 180,E1 -24969.52,E2 -24969.52} C_VEL
LIN {X 0,Y 163.876,Z 353.672,A -85,B 0,C 180,E1 -24972.465,E2 -24972.465} C_VEL
LIN {X 0,Y 167.045,Z 346.186,A -85,B 0,C 180,E1 -24975.66,E2 -24975.66} C_VEL
LIN {X 0,Y 169.074,Z 339.728,A -85,B 0,C 180,E1 -24978.434,E2 -24978.434} C_VEL
LIN {X 0,Y 169.329,Z 337.084,A -85,B 0,C 180,E1 -24979.874,E2 -24979.874} C_VEL
LIN {X 0,Y 168.966,Z 332.345,A -85,B 0,C 180,E1 -24983.092,E2 -24983.092} C_VEL
LIN {X 0,Y 168.41,Z 327.385,A -85,B 0,C 180,E1 -24987.141,E2 -24987.141} C_VEL
LIN {X 0,Y 168.01,Z 324.848,A -85,B 0,C 180,E1 -24989.865,E2 -24989.865} C_VEL
LIN {X 0,Y 167.719,Z 320.869,A -85,B 0,C 180,E1 -24995.222,E2 -24995.222} C_VEL
LIN {X 0,Y 167.583,Z 319.815,A -85,B 0,C 180,E1 -24998.385,E2 -24998.385} C_VEL
LIN {X 0,Y 167.252,Z 320.102,A -85,B 0,C 180,E1 -25000.399,E2 -25000.399} C_VEL
LIN {X 0,Y 166.477,Z 321.419,A -85,B 0,C 180,E1 -25002.375,E2 -25002.375} C_VEL
LIN {X 0,Y 164.452,Z 326.258,A -85,B 0,C 180,E1 -25007.662,E2 -25007.662} C_VEL
LIN {X 0,Y 164.543,Z 326.995,A -85,B 0,C 180,E1 -25009.042,E2 -25009.042} C_VEL
LIN {X 0,Y 164.82,Z 327.435,A -85,B 0,C 180,E1 -25010.176,E2 -25010.176} C_VEL
LIN {X 0,Y 165.539,Z 331.059,A -85,B 0,C 180,E1 -25015.125,E2 -25015.125} C_VEL
LIN {X 0,Y 165.574,Z 335.075,A -85,B 0,C 180,E1 -25018.78,E2 -25018.78} C_VEL
LIN {X 0,Y 165.278,Z 338.2,A -85,B 0,C 180,E1 -25021.214,E2 -25021.214} C_VEL
LIN {X 0,Y 164.365,Z 341.947,A -85,B 0,C 180,E1 -25023.673,E2 -25023.673} C_VEL
LIN {X 0,Y 164.032,Z 342.979,A -85,B 0,C 180,E1 -25024.296,E2 -25024.296} C_VEL
LIN {X 0,Y 163.16,Z 344.431,A -85,B 0,C 180,E1 -25024.986,E2 -25024.986} C_VEL
LIN {X 0,Y 156.263,Z 352.52,A -85,B 0,C 180,E1 -25028.338,E2 -25028.338} C_VEL
LIN {X 0,Y 150.632,Z 358.28,A -85,B 0,C 180,E1 -25031.548,E2 -25031.548} C_VEL
LIN {X 0,Y 145.501,Z 362.926,A -85,B 0,C 180,E1 -25034.982,E2 -25034.982} C_VEL
LIN {X 0,Y 140.925,Z 366.566,A -85,B 0,C 180,E1 -25038.647,E2 -25038.647} C_VEL
LIN {X 0,Y 136.978,Z 369.298,A -85,B 0,C 180,E1 -25042.556,E2 -25042.556} C_VEL
LIN {X 0,Y 132.325,Z 371.798,A -85,B 0,C 180,E1 -25048.549,E2 -25048.549} C_VEL
LIN {X 0,Y 129.975,Z 372.49,A -85,B 0,C 180,E1 -25052.726,E2 -25052.726} C_VEL
LIN {X 0,Y 128.234,Z 372.452,A -85,B 0,C 180,E1 -25057.068,E2 -25057.068} C_VEL
LIN {X 0,Y 127.025,Z 371.652,A -85,B 0,C 180,E1 -25061.593,E2 -25061.593} C_VEL
LIN {X 0,Y 126.455,Z 370.014,A -85,B 0,C 180,E1 -25066.253,E2 -25066.253} C_VEL
LIN {X 0,Y 126.763,Z 366.454,A -85,B 0,C 180,E1 -25072.423,E2 -25072.423} C_VEL
LIN {X 0,Y 127.621,Z 363.115,A -85,B 0,C 180,E1 -25076.588,E2 -25076.588} C_VEL
LIN {X 0,Y 129.145,Z 357.76,A -85,B 0,C 180,E1 -25081.69,E2 -25081.69} C_VEL
LIN {X 0,Y 131.606,Z 350.433,A -85,B 0,C 180,E1 -25086.992,E2 -25086.992} C_VEL
LIN {X 0,Y 134.283,Z 342.727,A -85,B 0,C 180,E1 -25091.265,E2 -25091.265} C_VEL
LIN {X 0,Y 137.445,Z 333.692,A -85,B 0,C 180,E1 -25095.189,E2 -25095.189} C_VEL
LIN {X 0,Y 140.617,Z 324.113,A -85,B 0,C 180,E1 -25098.469,E2 -25098.469} C_VEL
LIN {X 0,Y 142.453,Z 318.005,A -85,B 0,C 180,E1 -25100.202,E2 -25100.202} C_VEL
LIN {X 0,Y 141.69,Z 310.009,A -85,B 0,C 180,E1 -25102.716,E2 -25102.716} C_VEL
LIN {X 0,Y 139.903,Z 299.091,A -85,B 0,C 180,E1 -25105.843,E2 -25105.843} C_VEL
LIN {X 0,Y 138.006,Z 291.961,A -85,B 0,C 180,E1 -25107.813,E2 -25107.813} C_VEL
LIN {X 0,Y 133.544,Z 280.173,A -85,B 0,C 180,E1 -25111.119,E2 -25111.119} C_VEL
LIN {X 0,Y 131.092,Z 275.672,A -85,B 0,C 180,E1 -25112.476,E2 -25112.476} C_VEL
LIN {X 0,Y 129.818,Z 273.119,A -85,B 0,C 180,E1 -25113.202,E2 -25113.202} C_VEL
LIN {X 0,Y 129.648,Z 272.334,A -85,B 0,C 180,E1 -25113.498,E2 -25113.498} C_VEL
LIN {X 0,Y 129.505,Z 272.356,A -85,B 0,C 180,E1 -25119.371,E2 -25119.371} C_VEL
LIN {X 0,Y 129.383,Z 272.363,A -85,B 0,C 180,E1 -25122.551,E2 -25122.551} C_VEL
LIN {X 0,Y 129.175,Z 272.39,A -85,B 0,C 180,E1 -25129.055,E2 -25129.055} C_VEL
LIN {X 0,Y 129.126,Z 272.407,A -85,B 0,C 180,E1 -25132.397,E2 -25132.397} C_VEL
LIN {X 0,Y 129.05,Z 272.411,A -85,B 0,C 180,E1 -25139.396,E2 -25139.396} C_VEL
LIN {X 0,Y 129.02,Z 272.402,A -85,B 0,C 180,E1 -25145.217,E2 -25145.217} C_VEL
LIN {X 0,Y 129.042,Z 272.412,A -85,B 0,C 180,E1 -25150.812,E2 -25150.812} C_VEL
LIN {X 0,Y 129.033,Z 272.403,A -85,B 0,C 180,E1 -25155.08,E2 -25155.08} C_VEL
LIN {X 0,Y 129.051,Z 272.399,A -85,B 0,C 180,E1 -25159.681,E2 -25159.681} C_VEL
LIN {X 0,Y 129.032,Z 272.41,A -85,B 0,C 180,E1 -25164.789,E2 -25164.789} C_VEL
LIN {X 0,Y 129.031,Z 272.39,A -85,B 0,C 180,E1 -25170.652,E2 -25170.652} C_VEL
LIN {X 0,Y 129.107,Z 272.402,A -85,B 0,C 180,E1 -25177.607,E2 -25177.607} C_VEL
LIN {X 0,Y 129.153,Z 272.38,A -85,B 0,C 180,E1 -25180.95,E2 -25180.95} C_VEL
LIN {X 0,Y 129.368,Z 272.369,A -85,B 0,C 180,E1 -25187.929,E2 -25187.929} C_VEL
LIN {X 0,Y 129.478,Z 272.354,A -85,B 0,C 180,E1 -25190.634,E2 -25190.634} C_VEL
LIN {X 0,Y 130.091,Z 272.279,A -85,B 0,C 180,E1 -25200.005,E2 -25200.005} C_VEL
LIN {X 0,Y 129.478,Z 272.351,A -85,B 0,C 180,E1 -25209.377,E2 -25209.377} C_VEL
LIN {X 0,Y 129.351,Z 272.372,A -85,B 0,C 180,E1 -25212.558,E2 -25212.558} C_VEL
LIN {X 0,Y 129.16,Z 272.394,A -85,B 0,C 180,E1 -25219.06,E2 -25219.06} C_VEL
LIN {X 0,Y 129.116,Z 272.402,A -85,B 0,C 180,E1 -25222.402,E2 -25222.402} C_VEL
LIN {X 0,Y 129.131,Z 272.533,A -85,B 0,C 180,E1 -25228.002,E2 -25228.002} C_VEL
LIN {X 0,Y 129.464,Z 274.994,A -85,B 0,C 180,E1 -25232.884,E2 -25232.884} C_VEL
LIN {X 0,Y 130.03,Z 277.985,A -85,B 0,C 180,E1 -25238.436,E2 -25238.436} C_VEL
LIN {X 0,Y 130.569,Z 280.527,A -85,B 0,C 180,E1 -25242.841,E2 -25242.841} C_VEL
LIN {X 0,Y 131.728,Z 283.98,A -85,B 0,C 180,E1 -25243.56,E2 -25243.56} C_VEL
LIN {X 0,Y 132.732,Z 286.181,A -85,B 0,C 180,E1 -25244.11,E2 -25244.11} C_VEL
LIN {X 0,Y 136.182,Z 295.296,A -85,B 0,C 180,E1 -25246.268,E2 -25246.268} C_VEL
LIN {X 0,Y 137.342,Z 300.394,A -85,B 0,C 180,E1 -25247.365,E2 -25247.365} C_VEL
LIN {X 0,Y 138.386,Z 312.993,A -85,B 0,C 180,E1 -25250.045,E2 -25250.045} C_VEL
LIN {X 0,Y 138.561,Z 324.196,A -85,B 0,C 180,E1 -25252.798,E2 -25252.798} C_VEL
LIN {X 0,Y 138.386,Z 335.219,A -85,B 0,C 180,E1 -25256.036,E2 -25256.036} C_VEL
LIN {X 0,Y 137.766,Z 344.698,A -85,B 0,C 180,E1 -25259.325,E2 -25259.325} C_VEL
LIN {X 0,Y 135.781,Z 351.361,A -85,B 0,C 180,E1 -25261.876,E2 -25261.876} C_VEL
LIN {X 0,Y 132.815,Z 359.804,A -85,B 0,C 180,E1 -25265.787,E2 -25265.787} C_VEL
LIN {X 0,Y 130.221,Z 367.329,A -85,B 0,C 180,E1 -25270.285,E2 -25270.285} C_VEL
LIN {X 0,Y 128.133,Z 374.267,A -85,B 0,C 180,E1 -25275.709,E2 -25275.709} C_VEL
LIN {X 0,Y 127.199,Z 378.846,A -85,B 0,C 180,E1 -25280.457,E2 -25280.457} C_VEL
LIN {X 0,Y 126.971,Z 382.226,A -85,B 0,C 180,E1 -25285.137,E2 -25285.137} C_VEL
LIN {X 0,Y 127.041,Z 384.662,A -85,B 0,C 180,E1 -25289.998,E2 -25289.998} C_VEL
LIN {X 0,Y 126.806,Z 385.84,A -85,B 0,C 180,E1 -25293.891,E2 -25293.891} C_VEL
LIN {X 0,Y 126.972,Z 386.494,A -85,B 0,C 180,E1 -25299.557,E2 -25299.557} C_VEL
LIN {X 0,Y 128.427,Z 385.838,A -85,B 0,C 180,E1 -25305.878,E2 -25305.878} C_VEL
LIN {X 0,Y 129.704,Z 384.973,A -85,B 0,C 180,E1 -25308.97,E2 -25308.97} C_VEL
LIN {X 0,Y 133.581,Z 382.097,A -85,B 0,C 180,E1 -25314.889,E2 -25314.889} C_VEL
LIN {X 0,Y 138.841,Z 377.675,A -85,B 0,C 180,E1 -25320.408,E2 -25320.408} C_VEL
LIN {X 0,Y 143.481,Z 373.228,A -85,B 0,C 180,E1 -25324.282,E2 -25324.282} C_VEL
LIN {X 0,Y 149.924,Z 366.724,A -85,B 0,C 180,E1 -25328.396,E2 -25328.396} C_VEL
LIN {X 0,Y 153.886,Z 362.24,A -85,B 0,C 180,E1 -25330.6,E2 -25330.6} C_VEL
LIN {X 0,Y 157.858,Z 356.22,A -85,B 0,C 180,E1 -25333.514,E2 -25333.514} C_VEL
LIN {X 0,Y 161.44,Z 349.085,A -85,B 0,C 180,E1 -25336.815,E2 -25336.815} C_VEL
LIN {X 0,Y 163.793,Z 343.069,A -85,B 0,C 180,E1 -25339.602,E2 -25339.602} C_VEL
LIN {X 0,Y 164.098,Z 340.744,A -85,B 0,C 180,E1 -25341.026,E2 -25341.026} C_VEL
LIN {X 0,Y 164.04,Z 336.179,A -85,B 0,C 180,E1 -25344.488,E2 -25344.488} C_VEL
LIN {X 0,Y 163.787,Z 331.235,A -85,B 0,C 180,E1 -25349.111,E2 -25349.111} C_VEL
LIN {X 0,Y 163.56,Z 327.295,A -85,B 0,C 180,E1 -25354.548,E2 -25354.548} C_VEL
LIN {X 0,Y 163.588,Z 325.992,A -85,B 0,C 180,E1 -25357.249,E2 -25357.249} C_VEL
LIN {X 0,Y 163.927,Z 325.064,A -85,B 0,C 180,E1 -25362.532,E2 -25362.532} C_VEL
LIN {X 0,Y 164.069,Z 325.578,A -85,B 0,C 180,E1 -25365.103,E2 -25365.103} C_VEL
LIN {X 0,Y 164.543,Z 326.995,A -85,B 0,C 180,E1 -25369.042,E2 -25369.042} C_VEL
LIN {X 0,Y 164.646,Z 327.819,A -85,B 0,C 180,E1 -25370.38,E2 -25370.38} C_VEL
LIN {X 0,Y 164.17,Z 329.968,A -85,B 0,C 180,E1 -25372.298,E2 -25372.298} C_VEL
LIN {X 0,Y 163.151,Z 332.756,A -85,B 0,C 180,E1 -25374.113,E2 -25374.113} C_VEL
LIN {X 0,Y 160.584,Z 338.835,A -85,B 0,C 180,E1 -25377.796,E2 -25377.796} C_VEL
LIN {X 0,Y 160.092,Z 340.562,A -85,B 0,C 180,E1 -25379.112,E2 -25379.112} C_VEL
LIN {X 0,Y 159.463,Z 343.243,A -85,B 0,C 180,E1 -25381.258,E2 -25381.258} C_VEL
LIN {X 0,Y 158.803,Z 345.023,A -85,B 0,C 180,E1 -25382.532,E2 -25382.532} C_VEL
LIN {X 0,Y 157.549,Z 347.011,A -85,B 0,C 180,E1 -25383.562,E2 -25383.562} C_VEL
LIN {X 0,Y 151.396,Z 353.683,A -85,B 0,C 180,E1 -25386.461,E2 -25386.461} C_VEL
LIN {X 0,Y 144.432,Z 360.184,A -85,B 0,C 180,E1 -25390.323,E2 -25390.323} C_VEL
LIN {X 0,Y 137.82,Z 365.437,A -85,B 0,C 180,E1 -25394.767,E2 -25394.767} C_VEL
LIN {X 0,Y 131.505,Z 369.639,A -85,B 0,C 180,E1 -25400.32,E2 -25400.32} C_VEL
LIN {X 0,Y 126.395,Z 372.163,A -85,B 0,C 180,E1 -25406.406,E2 -25406.406} C_VEL
LIN {X 0,Y 123.414,Z 372.975,A -85,B 0,C 180,E1 -25411.333,E2 -25411.333} C_VEL
LIN {X 0,Y 121.468,Z 372.905,A -85,B 0,C 180,E1 -25415.905,E2 -25415.905} C_VEL
LIN {X 0,Y 120.131,Z 372.125,A -85,B 0,C 180,E1 -25420.492,E2 -25420.492} C_VEL
LIN {X 0,Y 119.326,Z 369.587,A -85,B 0,C 180,E1 -25427.368,E2 -25427.368} C_VEL
LIN {X 0,Y 119.96,Z 365.423,A -85,B 0,C 180,E1 -25434.138,E2 -25434.138} C_VEL
LIN {X 0,Y 120.988,Z 361.762,A -85,B 0,C 180,E1 -25438.482,E2 -25438.482} C_VEL
LIN {X 0,Y 122.984,Z 355.398,A -85,B 0,C 180,E1 -25444.201,E2 -25444.201} C_VEL
LIN {X 0,Y 125.804,Z 347.522,A -85,B 0,C 180,E1 -25449.566,E2 -25449.566} C_VEL
LIN {X 0,Y 129.016,Z 338.558,A -85,B 0,C 180,E1 -25454.197,E2 -25454.197} C_VEL
LIN {X 0,Y 132.641,Z 328.51,A -85,B 0,C 180,E1 -25458.192,E2 -25458.192} C_VEL
LIN {X 0,Y 135.605,Z 319.358,A -85,B 0,C 180,E1 -25461.057,E2 -25461.057} C_VEL
LIN {X 0,Y 135.223,Z 312.639,A -85,B 0,C 180,E1 -25463.286,E2 -25463.286} C_VEL
LIN {X 0,Y 133.773,Z 302.465,A -85,B 0,C 180,E1 -25466.465,E2 -25466.465} C_VEL
LIN {X 0,Y 132.22,Z 295.822,A -85,B 0,C 180,E1 -25468.48,E2 -25468.48} C_VEL
LIN {X 0,Y 128.056,Z 284.155,A -85,B 0,C 180,E1 -25472.008,E2 -25472.008} C_VEL
LIN {X 0,Y 123.895,Z 276.592,A -85,B 0,C 180,E1 -25474.59,E2 -25474.59} C_VEL
LIN {X 0,Y 122.636,Z 274.122,A -85,B 0,C 180,E1 -25475.397,E2 -25475.397} C_VEL
LIN {X 0,Y 122.476,Z 273.226,A -85,B 0,C 180,E1 -25475.662,E2 -25475.662} C_VEL
LIN {X 0,Y 122.435,Z 273.235,A -85,B 0,C 180,E1 -25479.918,E2 -25479.918} C_VEL
LIN {X 0,Y 122.276,Z 273.252,A -85,B 0,C 180,E1 -25483.293,E2 -25483.293} C_VEL
LIN {X 0,Y 122.064,Z 273.281,A -85,B 0,C 180,E1 -25490.212,E2 -25490.212} C_VEL
LIN {X 0,Y 121.987,Z 273.295,A -85,B 0,C 180,E1 -25493.786,E2 -25493.786} C_VEL
LIN {X 0,Y 121.949,Z 273.297,A -85,B 0,C 180,E1 -25500.191,E2 -25500.191} C_VEL
LIN {X 0,Y 121.942,Z 273.279,A -85,B 0,C 180,E1 -25506.219,E2 -25506.219} C_VEL
LIN {X 0,Y 121.962,Z 273.293,A -85,B 0,C 180,E1 -25511.495,E2 -25511.495} C_VEL
LIN {X 0,Y 121.967,Z 273.272,A -85,B 0,C 180,E1 -25518.514,E2 -25518.514} C_VEL
LIN {X 0,Y 121.983,Z 273.288,A -85,B 0,C 180,E1 -25524.827,E2 -25524.827} C_VEL
LIN {X 0,Y 121.94,Z 273.271,A -85,B 0,C 180,E1 -25529.832,E2 -25529.832} C_VEL
LIN {X 0,Y 121.982,Z 273.291,A -85,B 0,C 180,E1 -25536.221,E2 -25536.221} C_VEL
LIN {X 0,Y 122.044,Z 273.271,A -85,B 0,C 180,E1 -25539.793,E2 -25539.793} C_VEL
LIN {X 0,Y 122.24,Z 273.254,A -85,B 0,C 180,E1 -25546.71,E2 -25546.71} C_VEL
LIN {X 0,Y 122.408,Z 273.237,A -85,B 0,C 180,E1 -25550.087,E2 -25550.087} C_VEL
LIN {X 0,Y 122.598,Z 273.195,A -85,B 0,C 180,E1 -25556.719,E2 -25556.719} C_VEL
LIN {X 0,Y 123.044,Z 273.157,A -85,B 0,C 180,E1 -25560.005,E2 -25560.005} C_VEL
LIN {X 0,Y 122.424,Z 273.216,A -85,B 0,C 180,E1 -25566.598,E2 -25566.598} C_VEL
LIN {X 0,Y 122.414,Z 273.233,A -85,B 0,C 180,E1 -25569.923,E2 -25569.923} C_VEL
LIN {X 0,Y 122.246,Z 273.255,A -85,B 0,C 180,E1 -25573.3,E2 -25573.3} C_VEL
LIN {X 0,Y 122.053,Z 273.281,A -85,B 0,C 180,E1 -25580.217,E2 -25580.217} C_VEL
LIN {X 0,Y 122.104,Z 273.46,A -85,B 0,C 180,E1 -25587.422,E2 -25587.422} C_VEL
LIN {X 0,Y 122.283,Z 275.239,A -85,B 0,C 180,E1 -25591.154,E2 -25591.154} C_VEL
LIN {X 0,Y 122.787,Z 278.026,A -85,B 0,C 180,E1 -25596.741,E2 -25596.741} C_VEL
LIN {X 0,Y 123.243,Z 280.042,A -85,B 0,C 180,E1 -25600.54,E2 -25600.54} C_VEL
LIN {X 0,Y 124.367,Z 283.399,A -85,B 0,C 180,E1 -25601.294,E2 -25601.294} C_VEL
LIN {X 0,Y 128.317,Z 292.649,A -85,B 0,C 180,E1 -25603.754,E2 -25603.754} C_VEL
LIN {X 0,Y 130.706,Z 299.973,A -85,B 0,C 180,E1 -25605.651,E2 -25605.651} C_VEL
LIN {X 0,Y 131.673,Z 309.332,A -85,B 0,C 180,E1 -25607.766,E2 -25607.766} C_VEL
LIN {X 0,Y 132.003,Z 321.099,A -85,B 0,C 180,E1 -25610.724,E2 -25610.724} C_VEL
LIN {X 0,Y 131.682,Z 332.375,A -85,B 0,C 180,E1 -25614.048,E2 -25614.048} C_VEL
LIN {X 0,Y 131.194,Z 341.295,A -85,B 0,C 180,E1 -25617.152,E2 -25617.152} C_VEL
LIN {X 0,Y 130.721,Z 345.968,A -85,B 0,C 180,E1 -25618.97,E2 -25618.97} C_VEL
LIN {X 0,Y 127.422,Z 355.216,A -85,B 0,C 180,E1 -25622.931,E2 -25622.931} C_VEL
LIN {X 0,Y 124.412,Z 363.566,A -85,B 0,C 180,E1 -25627.584,E2 -25627.584} C_VEL
LIN {X 0,Y 122.399,Z 369.254,A -85,B 0,C 180,E1 -25631.589,E2 -25631.589} C_VEL
LIN {X 0,Y 120.83,Z 374.803,A -85,B 0,C 180,E1 -25636.545,E2 -25636.545} C_VEL
LIN {X 0,Y 120.011,Z 379.134,A -85,B 0,C 180,E1 -25641.58,E2 -25641.58} C_VEL
LIN {X 0,Y 119.893,Z 382.366,A -85,B 0,C 180,E1 -25646.638,E2 -25646.638} C_VEL
LIN {X 0,Y 119.98,Z 383.922,A -85,B 0,C 180,E1 -25649.998,E2 -25649.998} C_VEL
LIN {X 0,Y 119.741,Z 385.12,A -85,B 0,C 180,E1 -25653.74,E2 -25653.74} C_VEL
LIN {X 0,Y 119.954,Z 386.021,A -85,B 0,C 180,E1 -25660.121,E2 -25660.121} C_VEL
LIN {X 0,Y 121.584,Z 385.507,A -85,B 0,C 180,E1 -25666.797,E2 -25666.797} C_VEL
LIN {X 0,Y 124.91,Z 383.581,A -85,B 0,C 180,E1 -25673.192,E2 -25673.192} C_VEL
LIN {X 0,Y 127.144,Z 382.068,A -85,B 0,C 180,E1 -25676.243,E2 -25676.243} C_VEL
LIN {X 0,Y 132.744,Z 377.821,A -85,B 0,C 180,E1 -25681.966,E2 -25681.966} C_VEL
LIN {X 0,Y 139.505,Z 371.971,A -85,B 0,C 180,E1 -25687.193,E2 -25687.193} C_VEL
LIN {X 0,Y 146.558,Z 365.216,A -85,B 0,C 180,E1 -25691.249,E2 -25691.249} C_VEL
LIN {X 0,Y 149.458,Z 361.863,A -85,B 0,C 180,E1 -25692.985,E2 -25692.985} C_VEL
LIN {X 0,Y 153.894,Z 355.318,A -85,B 0,C 180,E1 -25696.337,E2 -25696.337} C_VEL
LIN {X 0,Y 157.264,Z 349.038,A -85,B 0,C 180,E1 -25699.437,E2 -25699.437} C_VEL
LIN {X 0,Y 158.207,Z 346.944,A -85,B 0,C 180,E1 -25700.48,E2 -25700.48} C_VEL
LIN {X 0,Y 158.71,Z 345.014,A -85,B 0,C 180,E1 -25701.683,E2 -25701.683} C_VEL
LIN {X 0,Y 158.971,Z 341.071,A -85,B 0,C 180,E1 -25704.915,E2 -25704.915} C_VEL
LIN {X 0,Y 159.085,Z 336.79,A -85,B 0,C 180,E1 -25709.151,E2 -25709.151} C_VEL
LIN {X 0,Y 159.054,Z 333.515,A -85,B 0,C 180,E1 -25713.773,E2 -25713.773} C_VEL
LIN {X 0,Y 159.287,Z 331.517,A -85,B 0,C 180,E1 -25717.899,E2 -25717.899} C_VEL
LIN {X 0,Y 159.562,Z 330.764,A -85,B 0,C 180,E1 -25722.038,E2 -25722.038} C_VEL
LIN {X 0,Y 159.695,Z 331.322,A -85,B 0,C 180,E1 -25725.504,E2 -25725.504} C_VEL
LIN {X 0,Y 160.206,Z 332.792,A -85,B 0,C 180,E1 -25729.89,E2 -25729.89} C_VEL
LIN {X 0,Y 160.353,Z 334.37,A -85,B 0,C 180,E1 -25732.44,E2 -25732.44} C_VEL
LIN {X 0,Y 160.543,Z 336.258,A -85,B 0,C 180,E1 -25734.973,E2 -25734.973} C_VEL
LIN {X 0,Y 160.178,Z 340.127,A -85,B 0,C 180,E1 -25738.739,E2 -25738.739} C_VEL
LIN {X 0,Y 160.092,Z 340.562,A -85,B 0,C 180,E1 -25739.112,E2 -25739.112} C_VEL
LIN {X 0,Y 159.335,Z 342.17,A -85,B 0,C 180,E1 -25740.079,E2 -25740.079} C_VEL
LIN {X 0,Y 157.094,Z 344.999,A -85,B 0,C 180,E1 -25741.124,E2 -25741.124} C_VEL
LIN {X 0,Y 149.076,Z 352.549,A -85,B 0,C 180,E1 -25743.362,E2 -25743.362} C_VEL
LIN {X 0,Y 148.287,Z 353.299,A -85,B 0,C 180,E1 -25743.699,E2 -25743.699} C_VEL
LIN {X 0,Y 141.63,Z 359.324,A -85,B 0,C 180,E1 -25747.061,E2 -25747.061} C_VEL
LIN {X 0,Y 135.806,Z 363.898,A -85,B 0,C 180,E1 -25750.51,E2 -25750.51} C_VEL
LIN {X 0,Y 128.536,Z 368.705,A -85,B 0,C 180,E1 -25755.86,E2 -25755.86} C_VEL
LIN {X 0,Y 124.319,Z 370.998,A -85,B 0,C 180,E1 -25759.822,E2 -25759.822} C_VEL
LIN {X 0,Y 120.681,Z 372.527,A -85,B 0,C 180,E1 -25764.051,E2 -25764.051} C_VEL
LIN {X 0,Y 117.636,Z 373.357,A -85,B 0,C 180,E1 -25768.545,E2 -25768.545} C_VEL
LIN {X 0,Y 115.268,Z 373.48,A -85,B 0,C 180,E1 -25773.273,E2 -25773.273} C_VEL
LIN {X 0,Y 113.548,Z 372.821,A -85,B 0,C 180,E1 -25778.231,E2 -25778.231} C_VEL
LIN {X 0,Y 112.484,Z 371.345,A -85,B 0,C 180,E1 -25783.406,E2 -25783.406} C_VEL
LIN {X 0,Y 112.242,Z 368.999,A -85,B 0,C 180,E1 -25788.7,E2 -25788.7} C_VEL
LIN {X 0,Y 112.825,Z 365.678,A -85,B 0,C 180,E1 -25794.064,E2 -25794.064} C_VEL
LIN {X 0,Y 114.111,Z 361.133,A -85,B 0,C 180,E1 -25799.557,E2 -25799.557} C_VEL
LIN {X 0,Y 116.154,Z 355.056,A -85,B 0,C 180,E1 -25805.158,E2 -25805.158} C_VEL
LIN {X 0,Y 118.7,Z 348.253,A -85,B 0,C 180,E1 -25810.017,E2 -25810.017} C_VEL
LIN {X 0,Y 121.938,Z 339.712,A -85,B 0,C 180,E1 -25814.749,E2 -25814.749} C_VEL
LIN {X 0,Y 125.808,Z 329.338,A -85,B 0,C 180,E1 -25819.134,E2 -25819.134} C_VEL
LIN {X 0,Y 128.719,Z 320.917,A -85,B 0,C 180,E1 -25821.918,E2 -25821.918} C_VEL
LIN {X 0,Y 129.034,Z 318.946,A -85,B 0,C 180,E1 -25822.569,E2 -25822.569} C_VEL
LIN {X 0,Y 128.055,Z 309.03,A -85,B 0,C 180,E1 -25826.052,E2 -25826.052} C_VEL
LIN {X 0,Y 126.512,Z 300.11,A -85,B 0,C 180,E1 -25828.949,E2 -25828.949} C_VEL
LIN {X 0,Y 122.42,Z 287.863,A -85,B 0,C 180,E1 -25833.025,E2 -25833.025} C_VEL
LIN {X 0,Y 117.448,Z 278.42,A -85,B 0,C 180,E1 -25836.551,E2 -25836.551} C_VEL
LIN {X 0,Y 115.64,Z 275.375,A -85,B 0,C 180,E1 -25837.751,E2 -25837.751} C_VEL
LIN {X 0,Y 115.359,Z 274.113,A -85,B 0,C 180,E1 -25838.101,E2 -25838.101} C_VEL
LIN {X 0,Y 115.294,Z 274.119,A -85,B 0,C 180,E1 -25842.788,E2 -25842.788} C_VEL
LIN {X 0,Y 115.023,Z 274.154,A -85,B 0,C 180,E1 -25847.79,E2 -25847.79} C_VEL
LIN {X 0,Y 114.957,Z 274.171,A -85,B 0,C 180,E1 -25853.519,E2 -25853.519} C_VEL
LIN {X 0,Y 114.871,Z 274.18,A -85,B 0,C 180,E1 -25861.082,E2 -25861.082} C_VEL
LIN {X 0,Y 114.874,Z 274.162,A -85,B 0,C 180,E1 -25867.722,E2 -25867.722} C_VEL
LIN {X 0,Y 114.88,Z 274.174,A -85,B 0,C 180,E1 -25872.776,E2 -25872.776} C_VEL
LIN {X 0,Y 114.89,Z 274.15,A -85,B 0,C 180,E1 -25877.718,E2 -25877.718} C_VEL
LIN {X 0,Y 114.896,Z 274.173,A -85,B 0,C 180,E1 -25882.676,E2 -25882.676} C_VEL
LIN {X 0,Y 114.868,Z 274.153,A -85,B 0,C 180,E1 -25888.937,E2 -25888.937} C_VEL
LIN {X 0,Y 114.946,Z 274.166,A -85,B 0,C 180,E1 -25896.514,E2 -25896.514} C_VEL
LIN {X 0,Y 115.011,Z 274.133,A -85,B 0,C 180,E1 -25902.216,E2 -25902.216} C_VEL
LIN {X 0,Y 115.253,Z 274.125,A -85,B 0,C 180,E1 -25907.34,E2 -25907.34} C_VEL
LIN {X 0,Y 115.366,Z 274.101,A -85,B 0,C 180,E1 -25913.008,E2 -25913.008} C_VEL
LIN {X 0,Y 115.996,Z 274.034,A -85,B 0,C 180,E1 -25920.006,E2 -25920.006} C_VEL
LIN {X 0,Y 115.366,Z 274.095,A -85,B 0,C 180,E1 -25927.004,E2 -25927.004} C_VEL
LIN {X 0,Y 115.255,Z 274.128,A -85,B 0,C 180,E1 -25932.664,E2 -25932.664} C_VEL
LIN {X 0,Y 115.018,Z 274.149,A -85,B 0,C 180,E1 -25937.795,E2 -25937.795} C_VEL
LIN {X 0,Y 114.955,Z 274.166,A -85,B 0,C 180,E1 -25943.497,E2 -25943.497} C_VEL
LIN {X 0,Y 114.99,Z 274.178,A -85,B 0,C 180,E1 -25946.308,E2 -25946.308} C_VEL
LIN {X 0,Y 115.383,Z 277.338,A -85,B 0,C 180,E1 -25953.249,E2 -25953.249} C_VEL
LIN {X 0,Y 115.882,Z 279.55,A -85,B 0,C 180,E1 -25957.851,E2 -25957.851} C_VEL
LIN {X 0,Y 116.933,Z 282.715,A -85,B 0,C 180,E1 -25958.653,E2 -25958.653} C_VEL
LIN {X 0,Y 118.162,Z 285.045,A -85,B 0,C 180,E1 -25959.433,E2 -25959.433} C_VEL
LIN {X 0,Y 122.742,Z 296.665,A -85,B 0,C 180,E1 -25962.838,E2 -25962.838} C_VEL
LIN {X 0,Y 124.782,Z 303.522,A -85,B 0,C 180,E1 -25964.758,E2 -25964.758} C_VEL
LIN {X 0,Y 125.445,Z 314.133,A -85,B 0,C 180,E1 -25967.399,E2 -25967.399} C_VEL
LIN {X 0,Y 125.358,Z 324.719,A -85,B 0,C 180,E1 -25970.378,E2 -25970.378} C_VEL
LIN {X 0,Y 124.783,Z 336.285,A -85,B 0,C 180,E1 -25974.242,E2 -25974.242} C_VEL
LIN {X 0,Y 123.882,Z 345.954,A -85,B 0,C 180,E1 -25978.083,E2 -25978.083} C_VEL
LIN {X 0,Y 120.496,Z 355.008,A -85,B 0,C 180,E1 -25982.184,E2 -25982.184} C_VEL
LIN {X 0,Y 117.378,Z 363.304,A -85,B 0,C 180,E1 -25987.094,E2 -25987.094} C_VEL
LIN {X 0,Y 114.956,Z 369.953,A -85,B 0,C 180,E1 -25992.199,E2 -25992.199} C_VEL
LIN {X 0,Y 113.52,Z 375.272,A -85,B 0,C 180,E1 -25997.484,E2 -25997.484} C_VEL
LIN {X 0,Y 112.875,Z 379.386,A -85,B 0,C 180,E1 -26002.845,E2 -26002.845} C_VEL
LIN {X 0,Y 112.835,Z 381.538,A -85,B 0,C 180,E1 -26006.427,E2 -26006.427} C_VEL
LIN {X 0,Y 112.92,Z 383.181,A -85,B 0,C 180,E1 -26009.998,E2 -26009.998} C_VEL
LIN {X 0,Y 112.7,Z 384.384,A -85,B 0,C 180,E1 -26013.754,E2 -26013.754} C_VEL
LIN {X 0,Y 112.962,Z 385.494,A -85,B 0,C 180,E1 -26020.755,E2 -26020.755} C_VEL
LIN {X 0,Y 114.759,Z 385.179,A -85,B 0,C 180,E1 -26027.829,E2 -26027.829} C_VEL
LIN {X 0,Y 118.398,Z 383.405,A -85,B 0,C 180,E1 -26034.549,E2 -26034.549} C_VEL
LIN {X 0,Y 123.654,Z 380.207,A -85,B 0,C 180,E1 -26040.763,E2 -26040.763} C_VEL
LIN {X 0,Y 128.419,Z 376.753,A -85,B 0,C 180,E1 -26045.07,E2 -26045.07} C_VEL
LIN {X 0,Y 133.922,Z 372.351,A -85,B 0,C 180,E1 -26049.028,E2 -26049.028} C_VEL
LIN {X 0,Y 141.325,Z 365.916,A -85,B 0,C 180,E1 -26053.137,E2 -26053.137} C_VEL
LIN {X 0,Y 145.267,Z 361.585,A -85,B 0,C 180,E1 -26055.526,E2 -26055.526} C_VEL
LIN {X 0,Y 149.718,Z 355.371,A -85,B 0,C 180,E1 -26058.909,E2 -26058.909} C_VEL
LIN {X 0,Y 152.607,Z 350.451,A -85,B 0,C 180,E1 -26061.524,E2 -26061.524} C_VEL
LIN {X 0,Y 153.453,Z 347.8,A -85,B 0,C 180,E1 -26063.455,E2 -26063.455} C_VEL
LIN {X 0,Y 153.821,Z 344.305,A -85,B 0,C 180,E1 -26066.747,E2 -26066.747} C_VEL
LIN {X 0,Y 154.126,Z 341.404,A -85,B 0,C 180,E1 -26070.037,E2 -26070.037} C_VEL
LIN {X 0,Y 154.446,Z 337.85,A -85,B 0,C 180,E1 -26075.82,E2 -26075.82} C_VEL
LIN {X 0,Y 154.733,Z 336.75,A -85,B 0,C 180,E1 -26078.689,E2 -26078.689} C_VEL
LIN {X 0,Y 154.971,Z 336.204,A -85,B 0,C 180,E1 -26082.238,E2 -26082.238} C_VEL
LIN {X 0,Y 155.016,Z 336.408,A -85,B 0,C 180,E1 -26084.211,E2 -26084.211} C_VEL
LIN {X 0,Y 155.347,Z 337.909,A -85,B 0,C 180,E1 -26089.57,E2 -26089.57} C_VEL
LIN {X 0,Y 155.358,Z 340.831,A -85,B 0,C 180,E1 -26094.38,E2 -26094.38} C_VEL
LIN {X 0,Y 154.604,Z 344.532,A -85,B 0,C 180,E1 -26098.347,E2 -26098.347} C_VEL
LIN {X 0,Y 153.997,Z 346.385,A -85,B 0,C 180,E1 -26099.996,E2 -26099.996} C_VEL
LIN {X 0,Y 153.23,Z 348.099,A -85,B 0,C 180,E1 -26101.31,E2 -26101.31} C_VEL
LIN {X 0,Y 152.143,Z 349.405,A -85,B 0,C 180,E1 -26101.981,E2 -26101.981} C_VEL
LIN {X 0,Y 148.287,Z 353.299,A -85,B 0,C 180,E1 -26103.699,E2 -26103.699} C_VEL
LIN {X 0,Y 144.655,Z 356.429,A -85,B 0,C 180,E1 -26105.059,E2 -26105.059} C_VEL
LIN {X 0,Y 137.409,Z 361.273,A -85,B 0,C 180,E1 -26107.002,E2 -26107.002} C_VEL
LIN {X 0,Y 130.136,Z 365.439,A -85,B 0,C 180,E1 -26109.263,E2 -26109.263} C_VEL
LIN {X 0,Y 126.56,Z 367.448,A -85,B 0,C 180,E1 -26111.137,E2 -26111.137} C_VEL
LIN {X 0,Y 123.022,Z 369.454,A -85,B 0,C 180,E1 -26113.798,E2 -26113.798} C_VEL
LIN {X 0,Y 118.286,Z 371.744,A -85,B 0,C 180,E1 -26118.083,E2 -26118.083} C_VEL
LIN {X 0,Y 114.222,Z 373.232,A -85,B 0,C 180,E1 -26122.646,E2 -26122.646} C_VEL
LIN {X 0,Y 110.89,Z 373.914,A -85,B 0,C 180,E1 -26127.47,E2 -26127.47} C_VEL
LIN {X 0,Y 108.337,Z 373.863,A -85,B 0,C 180,E1 -26132.511,E2 -26132.511} C_VEL
LIN {X 0,Y 106.536,Z 373.1,A -85,B 0,C 180,E1 -26137.667,E2 -26137.667} C_VEL
LIN {X 0,Y 105.456,Z 371.605,A -85,B 0,C 180,E1 -26142.858,E2 -26142.858} C_VEL
LIN {X 0,Y 105.14,Z 369.389,A -85,B 0,C 180,E1 -26148.056,E2 -26148.056} C_VEL
LIN {X 0,Y 106,Z 364.734,A -85,B 0,C 180,E1 -26155.7,E2 -26155.7} C_VEL
LIN {X 0,Y 107.665,Z 359.379,A -85,B 0,C 180,E1 -26161.907,E2 -26161.907} C_VEL
LIN {X 0,Y 109.914,Z 353.146,A -85,B 0,C 180,E1 -26167.443,E2 -26167.443} C_VEL
LIN {X 0,Y 113.057,Z 345.285,A -85,B 0,C 180,E1 -26172.828,E2 -26172.828} C_VEL
LIN {X 0,Y 116.85,Z 335.617,A -85,B 0,C 180,E1 -26177.85,E2 -26177.85} C_VEL
LIN {X 0,Y 120.693,Z 325.59,A -85,B 0,C 180,E1 -26181.811,E2 -26181.811} C_VEL
LIN {X 0,Y 122.3,Z 320.786,A -85,B 0,C 180,E1 -26183.402,E2 -26183.402} C_VEL
LIN {X 0,Y 121.711,Z 312.061,A -85,B 0,C 180,E1 -26186.692,E2 -26186.692} C_VEL
LIN {X 0,Y 120.63,Z 304.187,A -85,B 0,C 180,E1 -26189.471,E2 -26189.471} C_VEL
LIN {X 0,Y 117.427,Z 293.371,A -85,B 0,C 180,E1 -26193.433,E2 -26193.433} C_VEL
LIN {X 0,Y 115.105,Z 288.253,A -85,B 0,C 180,E1 -26195.444,E2 -26195.444} C_VEL
LIN {X 0,Y 109.899,Z 278.637,A -85,B 0,C 180,E1 -26199.505,E2 -26199.505} C_VEL
LIN {X 0,Y 108.518,Z 276.039,A -85,B 0,C 180,E1 -26200.615,E2 -26200.615} C_VEL
LIN {X 0,Y 108.302,Z 274.99,A -85,B 0,C 180,E1 -26200.991,E2 -26200.991} C_VEL
LIN {X 0,Y 108.04,Z 275.034,A -85,B 0,C 180,E1 -26205.084,E2 -26205.084} C_VEL
LIN {X 0,Y 107.922,Z 275.049,A -85,B 0,C 180,E1 -26213.002,E2 -26213.002} C_VEL
LIN {X 0,Y 107.812,Z 275.059,A -85,B 0,C 180,E1 -26221.435,E2 -26221.435} C_VEL
LIN {X 0,Y 107.778,Z 275.05,A -85,B 0,C 180,E1 -26228.521,E2 -26228.521} C_VEL
LIN {X 0,Y 107.782,Z 275.04,A -85,B 0,C 180,E1 -26235.832,E2 -26235.832} C_VEL
LIN {X 0,Y 107.79,Z 275.055,A -85,B 0,C 180,E1 -26241.484,E2 -26241.484} C_VEL
LIN {X 0,Y 107.81,Z 275.033,A -85,B 0,C 180,E1 -26248.574,E2 -26248.574} C_VEL
LIN {X 0,Y 107.909,Z 275.042,A -85,B 0,C 180,E1 -26257.005,E2 -26257.005} C_VEL
LIN {X 0,Y 108.031,Z 275.01,A -85,B 0,C 180,E1 -26264.923,E2 -26264.923} C_VEL
LIN {X 0,Y 108.255,Z 275,A -85,B 0,C 180,E1 -26268.776,E2 -26268.776} C_VEL
LIN {X 0,Y 108.446,Z 274.954,A -85,B 0,C 180,E1 -26276.291,E2 -26276.291} C_VEL
LIN {X 0,Y 108.945,Z 274.912,A -85,B 0,C 180,E1 -26280.006,E2 -26280.006} C_VEL
LIN {X 0,Y 108.306,Z 274.975,A -85,B 0,C 180,E1 -26287.463,E2 -26287.463} C_VEL
LIN {X 0,Y 108.177,Z 275.009,A -85,B 0,C 180,E1 -26292.956,E2 -26292.956} C_VEL
LIN {X 0,Y 107.911,Z 275.041,A -85,B 0,C 180,E1 -26299.011,E2 -26299.011} C_VEL
LIN {X 0,Y 107.959,Z 275.192,A -85,B 0,C 180,E1 -26305.868,E2 -26305.868} C_VEL
LIN {X 0,Y 108.323,Z 277.986,A -85,B 0,C 180,E1 -26312.492,E2 -26312.492} C_VEL
LIN {X 0,Y 108.452,Z 279.017,A -85,B 0,C 180,E1 -26314.76,E2 -26314.76} C_VEL
LIN {X 0,Y 109.542,Z 282.239,A -85,B 0,C 180,E1 -26315.7,E2 -26315.7} C_VEL
LIN {X 0,Y 110.993,Z 284.857,A -85,B 0,C 180,E1 -26316.704,E2 -26316.704} C_VEL
LIN {X 0,Y 114.163,Z 292.109,A -85,B 0,C 180,E1 -26319.132,E2 -26319.132} C_VEL
LIN {X 0,Y 117.931,Z 303.101,A -85,B 0,C 180,E1 -26322.687,E2 -26322.687} C_VEL
LIN {X 0,Y 118.709,Z 307.144,A -85,B 0,C 180,E1 -26323.881,E2 -26323.881} C_VEL
LIN {X 0,Y 118.973,Z 317.839,A -85,B 0,C 180,E1 -26326.823,E2 -26326.823} C_VEL
LIN {X 0,Y 118.546,Z 329.272,A -85,B 0,C 180,E1 -26330.425,E2 -26330.425} C_VEL
LIN {X 0,Y 117.81,Z 339.831,A -85,B 0,C 180,E1 -26334.432,E2 -26334.432} C_VEL
LIN {X 0,Y 116.98,Z 346.336,A -85,B 0,C 180,E1 -26337.266,E2 -26337.266} C_VEL
LIN {X 0,Y 113.613,Z 354.8,A -85,B 0,C 180,E1 -26341.351,E2 -26341.351} C_VEL
LIN {X 0,Y 110.369,Z 363.044,A -85,B 0,C 180,E1 -26346.546,E2 -26346.546} C_VEL
LIN {X 0,Y 108.211,Z 368.65,A -85,B 0,C 180,E1 -26351.048,E2 -26351.048} C_VEL
LIN {X 0,Y 106.593,Z 374.128,A -85,B 0,C 180,E1 -26356.656,E2 -26356.656} C_VEL
LIN {X 0,Y 105.845,Z 378.397,A -85,B 0,C 180,E1 -26362.367,E2 -26362.367} C_VEL
LIN {X 0,Y 105.793,Z 380.625,A -85,B 0,C 180,E1 -26366.189,E2 -26366.189} C_VEL
LIN {X 0,Y 105.86,Z 382.388,A -85,B 0,C 180,E1 -26369.998,E2 -26369.998} C_VEL
LIN {X 0,Y 105.647,Z 383.641,A -85,B 0,C 180,E1 -26373.812,E2 -26373.812} C_VEL
LIN {X 0,Y 105.968,Z 384.942,A -85,B 0,C 180,E1 -26381.474,E2 -26381.474} C_VEL
LIN {X 0,Y 107.98,Z 384.814,A -85,B 0,C 180,E1 -26388.989,E2 -26388.989} C_VEL
LIN {X 0,Y 111.965,Z 383.253,A -85,B 0,C 180,E1 -26396.062,E2 -26396.062} C_VEL
LIN {X 0,Y 117.593,Z 380.221,A -85,B 0,C 180,E1 -26402.538,E2 -26402.538} C_VEL
LIN {X 0,Y 124.535,Z 375.689,A -85,B 0,C 180,E1 -26408.37,E2 -26408.37} C_VEL
LIN {X 0,Y 130.651,Z 371.175,A -85,B 0,C 180,E1 -26412.25,E2 -26412.25} C_VEL
LIN {X 0,Y 137.368,Z 365.598,A -85,B 0,C 180,E1 -26415.744,E2 -26415.744} C_VEL
LIN {X 0,Y 141.264,Z 361.36,A -85,B 0,C 180,E1 -26418.265,E2 -26418.265} C_VEL
LIN {X 0,Y 145.7,Z 355.601,A -85,B 0,C 180,E1 -26421.61,E2 -26421.61} C_VEL
LIN {X 0,Y 147.3,Z 353.15,A -85,B 0,C 180,E1 -26423.049,E2 -26423.049} C_VEL
LIN {X 0,Y 148.139,Z 350.584,A -85,B 0,C 180,E1 -26425.293,E2 -26425.293} C_VEL
LIN {X 0,Y 148.908,Z 346.462,A -85,B 0,C 180,E1 -26430.017,E2 -26430.017} C_VEL
LIN {X 0,Y 149.305,Z 343.52,A -85,B 0,C 180,E1 -26434.931,E2 -26434.931} C_VEL
LIN {X 0,Y 149.688,Z 342.207,A -85,B 0,C 180,E1 -26437.934,E2 -26437.934} C_VEL
LIN {X 0,Y 149.957,Z 341.537,A -85,B 0,C 180,E1 -26440.844,E2 -26440.844} C_VEL
LIN {X 0,Y 150.087,Z 341.48,A -85,B 0,C 180,E1 -26443.678,E2 -26443.678} C_VEL
LIN {X 0,Y 150.239,Z 342.774,A -85,B 0,C 180,E1 -26449.211,E2 -26449.211} C_VEL
LIN {X 0,Y 150.08,Z 344.102,A -85,B 0,C 180,E1 -26451.92,E2 -26451.92} C_VEL
LIN {X 0,Y 149.827,Z 345.854,A -85,B 0,C 180,E1 -26454.612,E2 -26454.612} C_VEL
LIN {X 0,Y 149.133,Z 348.107,A -85,B 0,C 180,E1 -26457.294,E2 -26457.294} C_VEL
LIN {X 0,Y 148.471,Z 349.567,A -85,B 0,C 180,E1 -26458.775,E2 -26458.775} C_VEL
LIN {X 0,Y 147.552,Z 351.091,A -85,B 0,C 180,E1 -26459.995,E2 -26459.995} C_VEL
LIN {X 0,Y 139.496,Z 358.313,A -85,B 0,C 180,E1 -26463.604,E2 -26463.604} C_VEL
LIN {X 0,Y 131.921,Z 364.011,A -85,B 0,C 180,E1 -26467.681,E2 -26467.681} C_VEL
LIN {X 0,Y 126.56,Z 367.448,A -85,B 0,C 180,E1 -26471.137,E2 -26471.137} C_VEL
LIN {X 0,Y 123.069,Z 369.26,A -85,B 0,C 180,E1 -26473.166,E2 -26473.166} C_VEL
LIN {X 0,Y 116.124,Z 371.8,A -85,B 0,C 180,E1 -26476.339,E2 -26476.339} C_VEL
LIN {X 0,Y 109.491,Z 373.564,A -85,B 0,C 180,E1 -26479.97,E2 -26479.97} C_VEL
LIN {X 0,Y 106.615,Z 374.154,A -85,B 0,C 180,E1 -26482.686,E2 -26482.686} C_VEL
LIN {X 0,Y 102.918,Z 374.453,A -85,B 0,C 180,E1 -26488.548,E2 -26488.548} C_VEL
LIN {X 0,Y 100.494,Z 373.918,A -85,B 0,C 180,E1 -26494.011,E2 -26494.011} C_VEL
LIN {X 0,Y 98.866,Z 372.623,A -85,B 0,C 180,E1 -26499.766,E2 -26499.766} C_VEL
LIN {X 0,Y 98.094,Z 370.482,A -85,B 0,C 180,E1 -26505.752,E2 -26505.752} C_VEL
LIN {X 0,Y 98.51,Z 366.302,A -85,B 0,C 180,E1 -26513.615,E2 -26513.615} C_VEL
LIN {X 0,Y 100.029,Z 361.159,A -85,B 0,C 180,E1 -26520.543,E2 -26520.543} C_VEL
LIN {X 0,Y 102.292,Z 355.05,A -85,B 0,C 180,E1 -26526.733,E2 -26526.733} C_VEL
LIN {X 0,Y 105.369,Z 347.499,A -85,B 0,C 180,E1 -26532.536,E2 -26532.536} C_VEL
LIN {X 0,Y 109.162,Z 338.397,A -85,B 0,C 180,E1 -26537.86,E2 -26537.86} C_VEL
LIN {X 0,Y 112.706,Z 329.73,A -85,B 0,C 180,E1 -26541.757,E2 -26541.757} C_VEL
LIN {X 0,Y 115.755,Z 321.357,A -85,B 0,C 180,E1 -26544.777,E2 -26544.777} C_VEL
LIN {X 0,Y 115.021,Z 311.195,A -85,B 0,C 180,E1 -26548.889,E2 -26548.889} C_VEL
LIN {X 0,Y 113.978,Z 304.855,A -85,B 0,C 180,E1 -26551.328,E2 -26551.328} C_VEL
LIN {X 0,Y 111.223,Z 295.532,A -85,B 0,C 180,E1 -26555.043,E2 -26555.043} C_VEL
LIN {X 0,Y 105.782,Z 284.754,A -85,B 0,C 180,E1 -26560.044,E2 -26560.044} C_VEL
LIN {X 0,Y 103.195,Z 280.012,A -85,B 0,C 180,E1 -26562.312,E2 -26562.312} C_VEL
LIN {X 0,Y 101.423,Z 277.285,A -85,B 0,C 180,E1 -26563.784,E2 -26563.784} C_VEL
LIN {X 0,Y 101.048,Z 275.902,A -85,B 0,C 180,E1 -26564.267,E2 -26564.267} C_VEL
LIN {X 0,Y 100.827,Z 275.926,A -85,B 0,C 180,E1 -26570.399,E2 -26570.399} C_VEL
LIN {X 0,Y 100.765,Z 275.93,A -85,B 0,C 180,E1 -26574.963,E2 -26574.963} C_VEL
LIN {X 0,Y 100.707,Z 275.94,A -85,B 0,C 180,E1 -26583.143,E2 -26583.143} C_VEL
LIN {X 0,Y 100.72,Z 275.936,A -85,B 0,C 180,E1 -26589.877,E2 -26589.877} C_VEL
LIN {X 0,Y 100.747,Z 275.916,A -85,B 0,C 180,E1 -26595.776,E2 -26595.776} C_VEL
LIN {X 0,Y 100.73,Z 275.931,A -85,B 0,C 180,E1 -26601.111,E2 -26601.111} C_VEL
LIN {X 0,Y 100.71,Z 275.928,A -85,B 0,C 180,E1 -26606.871,E2 -26606.871} C_VEL
LIN {X 0,Y 100.785,Z 275.929,A -85,B 0,C 180,E1 -26615.274,E2 -26615.274} C_VEL
LIN {X 0,Y 100.815,Z 275.915,A -85,B 0,C 180,E1 -26619.608,E2 -26619.608} C_VEL
LIN {X 0,Y 101.103,Z 275.884,A -85,B 0,C 180,E1 -26626.71,E2 -26626.71} C_VEL
LIN {X 0,Y 101.244,Z 275.866,A -85,B 0,C 180,E1 -26632.026,E2 -26632.026} C_VEL
LIN {X 0,Y 101.868,Z 275.794,A -85,B 0,C 180,E1 -26640.007,E2 -26640.007} C_VEL
LIN {X 0,Y 101.245,Z 275.856,A -85,B 0,C 180,E1 -26647.987,E2 -26647.987} C_VEL
LIN {X 0,Y 101.107,Z 275.888,A -85,B 0,C 180,E1 -26653.299,E2 -26653.299} C_VEL
LIN {X 0,Y 100.847,Z 275.924,A -85,B 0,C 180,E1 -26662.545,E2 -26662.545} C_VEL
LIN {X 0,Y 100.908,Z 276.11,A -85,B 0,C 180,E1 -26665.116,E2 -26665.116} C_VEL
LIN {X 0,Y 101.244,Z 278.608,A -85,B 0,C 180,E1 -26671.236,E2 -26671.236} C_VEL
LIN {X 0,Y 102.383,Z 281.904,A -85,B 0,C 180,E1 -26672.339,E2 -26672.339} C_VEL
LIN {X 0,Y 103.756,Z 284.448,A -85,B 0,C 180,E1 -26673.464,E2 -26673.464} C_VEL
LIN {X 0,Y 107.381,Z 292.484,A -85,B 0,C 180,E1 -26676.615,E2 -26676.615} C_VEL
LIN {X 0,Y 111.379,Z 304.134,A -85,B 0,C 180,E1 -26680.779,E2 -26680.779} C_VEL
LIN {X 0,Y 112.498,Z 308.566,A -85,B 0,C 180,E1 -26682.316,E2 -26682.316} C_VEL
LIN {X 0,Y 112.508,Z 319.917,A -85,B 0,C 180,E1 -26685.742,E2 -26685.742} C_VEL
LIN {X 0,Y 111.825,Z 331.108,A -85,B 0,C 180,E1 -26689.639,E2 -26689.639} C_VEL
LIN {X 0,Y 110.837,Z 341.804,A -85,B 0,C 180,E1 -26694.087,E2 -26694.087} C_VEL
LIN {X 0,Y 110.012,Z 346.767,A -85,B 0,C 180,E1 -26696.426,E2 -26696.426} C_VEL
LIN {X 0,Y 106.144,Z 355.947,A -85,B 0,C 180,E1 -26701.31,E2 -26701.31} C_VEL
LIN {X 0,Y 102.858,Z 363.885,A -85,B 0,C 180,E1 -26706.864,E2 -26706.864} C_VEL
LIN {X 0,Y 100.763,Z 369.258,A -85,B 0,C 180,E1 -26711.705,E2 -26711.705} C_VEL
LIN {X 0,Y 99.297,Z 374.524,A -85,B 0,C 180,E1 -26717.739,E2 -26717.739} C_VEL
LIN {X 0,Y 98.809,Z 377.379,A -85,B 0,C 180,E1 -26721.819,E2 -26721.819} C_VEL
LIN {X 0,Y 98.742,Z 379.697,A -85,B 0,C 180,E1 -26725.916,E2 -26725.916} C_VEL
LIN {X 0,Y 98.801,Z 381.54,A -85,B 0,C 180,E1 -26729.998,E2 -26729.998} C_VEL
LIN {X 0,Y 98.584,Z 382.898,A -85,B 0,C 180,E1 -26734.086,E2 -26734.086} C_VEL
LIN {X 0,Y 99.007,Z 384.386,A -85,B 0,C 180,E1 -26742.293,E2 -26742.293} C_VEL
LIN {X 0,Y 101.256,Z 384.415,A -85,B 0,C 180,E1 -26750.304,E2 -26750.304} C_VEL
LIN {X 0,Y 105.606,Z 383.065,A -85,B 0,C 180,E1 -26757.762,E2 -26757.762} C_VEL
LIN {X 0,Y 111.652,Z 380.258,A -85,B 0,C 180,E1 -26764.505,E2 -26764.505} C_VEL
LIN {X 0,Y 119.045,Z 375.944,A -85,B 0,C 180,E1 -26770.494,E2 -26770.494} C_VEL
LIN {X 0,Y 125.512,Z 371.619,A -85,B 0,C 180,E1 -26774.419,E2 -26774.419} C_VEL
LIN {X 0,Y 132.52,Z 366.285,A -85,B 0,C 180,E1 -26777.939,E2 -26777.939} C_VEL
LIN {X 0,Y 136.581,Z 362.299,A -85,B 0,C 180,E1 -26780.517,E2 -26780.517} C_VEL
LIN {X 0,Y 141.272,Z 356.792,A -85,B 0,C 180,E1 -26783.937,E2 -26783.937} C_VEL
LIN {X 0,Y 141.975,Z 355.679,A -85,B 0,C 180,E1 -26784.76,E2 -26784.76} C_VEL
LIN {X 0,Y 142.966,Z 352.599,A -85,B 0,C 180,E1 -26788.247,E2 -26788.247} C_VEL
LIN {X 0,Y 143.492,Z 350.74,A -85,B 0,C 180,E1 -26790.669,E2 -26790.669} C_VEL
LIN {X 0,Y 143.906,Z 348.911,A -85,B 0,C 180,E1 -26793.921,E2 -26793.921} C_VEL
LIN {X 0,Y 144.408,Z 347.268,A -85,B 0,C 180,E1 -26797.617,E2 -26797.617} C_VEL
LIN {X 0,Y 144.757,Z 346.556,A -85,B 0,C 180,E1 -26800.128,E2 -26800.128} C_VEL
LIN {X 0,Y 144.88,Z 346.347,A -85,B 0,C 180,E1 -26803.074,E2 -26803.074} C_VEL
LIN {X 0,Y 144.87,Z 347.381,A -85,B 0,C 180,E1 -26808.806,E2 -26808.806} C_VEL
LIN {X 0,Y 144.612,Z 348.6,A -85,B 0,C 180,E1 -26811.612,E2 -26811.612} C_VEL
LIN {X 0,Y 144.122,Z 350.225,A -85,B 0,C 180,E1 -26814.399,E2 -26814.399} C_VEL
LIN {X 0,Y 143.095,Z 352.452,A -85,B 0,C 180,E1 -26817.18,E2 -26817.18} C_VEL
LIN {X 0,Y 142.533,Z 353.29,A -85,B 0,C 180,E1 -26818.061,E2 -26818.061} C_VEL
LIN {X 0,Y 133.609,Z 360.56,A -85,B 0,C 180,E1 -26822.006,E2 -26822.006} C_VEL
LIN {X 0,Y 125.323,Z 366.104,A -85,B 0,C 180,E1 -26826.434,E2 -26826.434} C_VEL
LIN {X 0,Y 119.617,Z 369.303,A -85,B 0,C 180,E1 -26830.146,E2 -26830.146} C_VEL
LIN {X 0,Y 114.451,Z 371.672,A -85,B 0,C 180,E1 -26834.212,E2 -26834.212} C_VEL
LIN {X 0,Y 109.954,Z 373.301,A -85,B 0,C 180,E1 -26838.631,E2 -26838.631} C_VEL
LIN {X 0,Y 106.615,Z 374.154,A -85,B 0,C 180,E1 -26842.686,E2 -26842.686} C_VEL
LIN {X 0,Y 103.961,Z 374.483,A -85,B 0,C 180,E1 -26845.554,E2 -26845.554} C_VEL
LIN {X 0,Y 98.449,Z 374.506,A -85,B 0,C 180,E1 -26850.224,E2 -26850.224} C_VEL
LIN {X 0,Y 94.347,Z 373.987,A -85,B 0,C 180,E1 -26854.274,E2 -26854.274} C_VEL
LIN {X 0,Y 92.284,Z 373.208,A -85,B 0,C 180,E1 -26857.658,E2 -26857.658} C_VEL
LIN {X 0,Y 91.911,Z 372.862,A -85,B 0,C 180,E1 -26858.85,E2 -26858.85} C_VEL
LIN {X 0,Y 90.979,Z 370.334,A -85,B 0,C 180,E1 -26865.957,E2 -26865.957} C_VEL
LIN {X 0,Y 91.161,Z 367.417,A -85,B 0,C 180,E1 -26871.924,E2 -26871.924} C_VEL
LIN {X 0,Y 92.502,Z 362.667,A -85,B 0,C 180,E1 -26879.149,E2 -26879.149} C_VEL
LIN {X 0,Y 94.77,Z 356.465,A -85,B 0,C 180,E1 -26886.214,E2 -26886.214} C_VEL
LIN {X 0,Y 97.614,Z 349.774,A -85,B 0,C 180,E1 -26892.033,E2 -26892.033} C_VEL
LIN {X 0,Y 101.607,Z 340.674,A -85,B 0,C 180,E1 -26898.026,E2 -26898.026} C_VEL
LIN {X 0,Y 105.308,Z 332.086,A -85,B 0,C 180,E1 -26902.332,E2 -26902.332} C_VEL
LIN {X 0,Y 108.959,Z 323.123,A -85,B 0,C 180,E1 -26905.841,E2 -26905.841} C_VEL
LIN {X 0,Y 109.087,Z 319.931,A -85,B 0,C 180,E1 -26907.222,E2 -26907.222} C_VEL
LIN {X 0,Y 108.292,Z 310.09,A -85,B 0,C 180,E1 -26911.398,E2 -26911.398} C_VEL
LIN {X 0,Y 105.912,Z 300.492,A -85,B 0,C 180,E1 -26915.6,E2 -26915.6} C_VEL
LIN {X 0,Y 102.961,Z 293.792,A -85,B 0,C 180,E1 -26918.935,E2 -26918.935} C_VEL
LIN {X 0,Y 98.676,Z 285.184,A -85,B 0,C 180,E1 -26923.387,E2 -26923.387} C_VEL
LIN {X 0,Y 95.784,Z 280.795,A -85,B 0,C 180,E1 -26926.138,E2 -26926.138} C_VEL
LIN {X 0,Y 94.122,Z 278.226,A -85,B 0,C 180,E1 -26927.801,E2 -26927.801} C_VEL
LIN {X 0,Y 93.763,Z 276.8,A -85,B 0,C 180,E1 -26928.437,E2 -26928.437} C_VEL
LIN {X 0,Y 93.661,Z 276.809,A -85,B 0,C 180,E1 -26935.802,E2 -26935.802} C_VEL
LIN {X 0,Y 93.617,Z 276.813,A -85,B 0,C 180,E1 -26944.345,E2 -26944.345} C_VEL
LIN {X 0,Y 93.642,Z 276.82,A -85,B 0,C 180,E1 -26952.493,E2 -26952.493} C_VEL
LIN {X 0,Y 93.645,Z 276.797,A -85,B 0,C 180,E1 -26958.636,E2 -26958.636} C_VEL
LIN {X 0,Y 93.624,Z 276.817,A -85,B 0,C 180,E1 -26965.666,E2 -26965.666} C_VEL
LIN {X 0,Y 93.668,Z 276.812,A -85,B 0,C 180,E1 -26974.212,E2 -26974.212} C_VEL
LIN {X 0,Y 93.692,Z 276.81,A -85,B 0,C 180,E1 -26977.98,E2 -26977.98} C_VEL
LIN {X 0,Y 94.023,Z 276.764,A -85,B 0,C 180,E1 -26986.35,E2 -26986.35} C_VEL
LIN {X 0,Y 94.177,Z 276.748,A -85,B 0,C 180,E1 -26991.424,E2 -26991.424} C_VEL
LIN {X 0,Y 94.794,Z 276.675,A -85,B 0,C 180,E1 -27000.007,E2 -27000.007} C_VEL
LIN {X 0,Y 94.179,Z 276.738,A -85,B 0,C 180,E1 -27008.59,E2 -27008.59} C_VEL
LIN {X 0,Y 94.027,Z 276.768,A -85,B 0,C 180,E1 -27013.66,E2 -27013.66} C_VEL
LIN {X 0,Y 93.851,Z 276.877,A -85,B 0,C 180,E1 -27023.998,E2 -27023.998} C_VEL
LIN {X 0,Y 93.952,Z 278.044,A -85,B 0,C 180,E1 -27026.976,E2 -27026.976} C_VEL
LIN {X 0,Y 94.972,Z 281.058,A -85,B 0,C 180,E1 -27028.156,E2 -27028.156} C_VEL
LIN {X 0,Y 96.659,Z 283.886,A -85,B 0,C 180,E1 -27029.699,E2 -27029.699} C_VEL
LIN {X 0,Y 100.796,Z 293.444,A -85,B 0,C 180,E1 -27033.911,E2 -27033.911} C_VEL
LIN {X 0,Y 103.491,Z 300.866,A -85,B 0,C 180,E1 -27036.994,E2 -27036.994} C_VEL
LIN {X 0,Y 106.246,Z 310.271,A -85,B 0,C 180,E1 -27040.723,E2 -27040.723} C_VEL
LIN {X 0,Y 106.188,Z 320.004,A -85,B 0,C 180,E1 -27043.903,E2 -27043.903} C_VEL
LIN {X 0,Y 105.376,Z 330.346,A -85,B 0,C 180,E1 -27047.711,E2 -27047.711} C_VEL
LIN {X 0,Y 104.166,Z 341.449,A -85,B 0,C 180,E1 -27052.608,E2 -27052.608} C_VEL
LIN {X 0,Y 103.11,Z 346.991,A -85,B 0,C 180,E1 -27055.412,E2 -27055.412} C_VEL
LIN {X 0,Y 99.292,Z 355.6,A -85,B 0,C 180,E1 -27060.297,E2 -27060.297} C_VEL
LIN {X 0,Y 95.841,Z 363.517,A -85,B 0,C 180,E1 -27066.212,E2 -27066.212} C_VEL
LIN {X 0,Y 93.368,Z 369.869,A -85,B 0,C 180,E1 -27072.475,E2 -27072.475} C_VEL
LIN {X 0,Y 92.033,Z 374.902,A -85,B 0,C 180,E1 -27078.992,E2 -27078.992} C_VEL
LIN {X 0,Y 91.684,Z 378.752,A -85,B 0,C 180,E1 -27085.601,E2 -27085.601} C_VEL
LIN {X 0,Y 91.744,Z 380.675,A -85,B 0,C 180,E1 -27089.998,E2 -27089.998} C_VEL
LIN {X 0,Y 91.541,Z 382.102,A -85,B 0,C 180,E1 -27094.401,E2 -27094.401} C_VEL
LIN {X 0,Y 92.081,Z 383.791,A -85,B 0,C 180,E1 -27103.234,E2 -27103.234} C_VEL
LIN {X 0,Y 94.597,Z 384.017,A -85,B 0,C 180,E1 -27111.804,E2 -27111.804} C_VEL
LIN {X 0,Y 99.343,Z 382.844,A -85,B 0,C 180,E1 -27119.681,E2 -27119.681} C_VEL
LIN {X 0,Y 105.845,Z 380.28,A -85,B 0,C 180,E1 -27126.695,E2 -27126.695} C_VEL
LIN {X 0,Y 111.641,Z 377.354,A -85,B 0,C 180,E1 -27131.373,E2 -27131.373} C_VEL
LIN {X 0,Y 118.176,Z 373.571,A -85,B 0,C 180,E1 -27135.53,E2 -27135.53} C_VEL
LIN {X 0,Y 125.484,Z 368.812,A -85,B 0,C 180,E1 -27139.118,E2 -27139.118} C_VEL
LIN {X 0,Y 127.853,Z 367.042,A -85,B 0,C 180,E1 -27140.312,E2 -27140.312} C_VEL
LIN {X 0,Y 133.298,Z 362.016,A -85,B 0,C 180,E1 -27143.719,E2 -27143.719} C_VEL
LIN {X 0,Y 136.053,Z 359.085,A -85,B 0,C 180,E1 -27145.738,E2 -27145.738} C_VEL
LIN {X 0,Y 137.328,Z 356.262,A -85,B 0,C 180,E1 -27149.213,E2 -27149.213} C_VEL
LIN {X 0,Y 138.089,Z 354.072,A -85,B 0,C 180,E1 -27152.734,E2 -27152.734} C_VEL
LIN {X 0,Y 138.618,Z 352.541,A -85,B 0,C 180,E1 -27156.066,E2 -27156.066} C_VEL
LIN {X 0,Y 139.192,Z 351.427,A -85,B 0,C 180,E1 -27159.297,E2 -27159.297} C_VEL
LIN {X 0,Y 139.461,Z 350.975,A -85,B 0,C 180,E1 -27163.226,E2 -27163.226} C_VEL
LIN {X 0,Y 139.29,Z 351.723,A -85,B 0,C 180,E1 -27168.352,E2 -27168.352} C_VEL
LIN {X 0,Y 138.945,Z 352.826,A -85,B 0,C 180,E1 -27171.267,E2 -27171.267} C_VEL
LIN {X 0,Y 138.189,Z 354.345,A -85,B 0,C 180,E1 -27174.157,E2 -27174.157} C_VEL
LIN {X 0,Y 137.59,Z 355.365,A -85,B 0,C 180,E1 -27175.601,E2 -27175.601} C_VEL
LIN {X 0,Y 135.454,Z 357.293,A -85,B 0,C 180,E1 -27177.021,E2 -27177.021} C_VEL
LIN {X 0,Y 126.515,Z 363.588,A -85,B 0,C 180,E1 -27180.908,E2 -27180.908} C_VEL
LIN {X 0,Y 117.913,Z 368.486,A -85,B 0,C 180,E1 -27185.543,E2 -27185.543} C_VEL
LIN {X 0,Y 110.019,Z 372.038,A -85,B 0,C 180,E1 -27191.042,E2 -27191.042} C_VEL
LIN {X 0,Y 103.156,Z 374.213,A -85,B 0,C 180,E1 -27197.488,E2 -27197.488} C_VEL
LIN {X 0,Y 99.008,Z 374.875,A -85,B 0,C 180,E1 -27202.669,E2 -27202.669} C_VEL
LIN {X 0,Y 95.699,Z 374.813,A -85,B 0,C 180,E1 -27208.21,E2 -27208.21} C_VEL
LIN {X 0,Y 93.265,Z 374.044,A -85,B 0,C 180,E1 -27214.018,E2 -27214.018} C_VEL
LIN {X 0,Y 91.911,Z 372.862,A -85,B 0,C 180,E1 -27218.85,E2 -27218.85} C_VEL
LIN {X 0,Y 90.602,Z 371.735,A -85,B 0,C 180,E1 -27222.39,E2 -27222.39} C_VEL
LIN {X 0,Y 87.4,Z 369.292,A -85,B 0,C 180,E1 -27228.218,E2 -27228.218} C_VEL
LIN {X 0,Y 85.311,Z 366.802,A -85,B 0,C 180,E1 -27233.054,E2 -27233.054} C_VEL
LIN {X 0,Y 84.873,Z 364.592,A -85,B 0,C 180,E1 -27236.767,E2 -27236.767} C_VEL
LIN {X 0,Y 85.054,Z 363.787,A -85,B 0,C 180,E1 -27237.993,E2 -27237.993} C_VEL
LIN {X 0,Y 86.993,Z 358.536,A -85,B 0,C 180,E1 -27244.868,E2 -27244.868} C_VEL
LIN {X 0,Y 90.001,Z 351.524,A -85,B 0,C 180,E1 -27251.802,E2 -27251.802} C_VEL
LIN {X 0,Y 93.543,Z 343.854,A -85,B 0,C 180,E1 -27257.571,E2 -27257.571} C_VEL
LIN {X 0,Y 97.922,Z 334.335,A -85,B 0,C 180,E1 -27262.996,E2 -27262.996} C_VEL
LIN {X 0,Y 102.591,Z 323.475,A -85,B 0,C 180,E1 -27267.548,E2 -27267.548} C_VEL
LIN {X 0,Y 102.144,Z 313.342,A -85,B 0,C 180,E1 -27272.304,E2 -27272.304} C_VEL
LIN {X 0,Y 100.149,Z 304.101,A -85,B 0,C 180,E1 -27276.753,E2 -27276.753} C_VEL
LIN {X 0,Y 97.633,Z 298.018,A -85,B 0,C 180,E1 -27280.068,E2 -27280.068} C_VEL
LIN {X 0,Y 94.253,Z 290.678,A -85,B 0,C 180,E1 -27284.256,E2 -27284.256} C_VEL
LIN {X 0,Y 92.102,Z 286.845,A -85,B 0,C 180,E1 -27286.76,E2 -27286.76} C_VEL
LIN {X 0,Y 90.275,Z 284.42,A -85,B 0,C 180,E1 -27288.643,E2 -27288.643} C_VEL
LIN {X 0,Y 89.109,Z 282.17,A -85,B 0,C 180,E1 -27290.109,E2 -27290.109} C_VEL
LIN {X 0,Y 87.172,Z 279.629,A -85,B 0,C 180,E1 -27292.259,E2 -27292.259} C_VEL
LIN {X 0,Y 86.6,Z 277.704,A -85,B 0,C 180,E1 -27293.308,E2 -27293.308} C_VEL
LIN {X 0,Y 86.477,Z 277.71,A -85,B 0,C 180,E1 -27299.187,E2 -27299.187} C_VEL
LIN {X 0,Y 86.545,Z 277.686,A -85,B 0,C 180,E1 -27305.716,E2 -27305.716} C_VEL
LIN {X 0,Y 86.567,Z 277.7,A -85,B 0,C 180,E1 -27313.07,E2 -27313.07} C_VEL
LIN {X 0,Y 86.567,Z 277.682,A -85,B 0,C 180,E1 -27319.508,E2 -27319.508} C_VEL
LIN {X 0,Y 86.574,Z 277.696,A -85,B 0,C 180,E1 -27325.381,E2 -27325.381} C_VEL
LIN {X 0,Y 86.584,Z 277.688,A -85,B 0,C 180,E1 -27333.241,E2 -27333.241} C_VEL
LIN {X 0,Y 86.645,Z 277.667,A -85,B 0,C 180,E1 -27341.076,E2 -27341.076} C_VEL
LIN {X 0,Y 86.932,Z 277.643,A -85,B 0,C 180,E1 -27345.972,E2 -27345.972} C_VEL
LIN {X 0,Y 87.086,Z 277.635,A -85,B 0,C 180,E1 -27350.72,E2 -27350.72} C_VEL
LIN {X 0,Y 87.72,Z 277.555,A -85,B 0,C 180,E1 -27360.008,E2 -27360.008} C_VEL
LIN {X 0,Y 87.088,Z 277.626,A -85,B 0,C 180,E1 -27369.296,E2 -27369.296} C_VEL
LIN {X 0,Y 86.938,Z 277.648,A -85,B 0,C 180,E1 -27374.043,E2 -27374.043} C_VEL
LIN {X 0,Y 86.728,Z 277.681,A -85,B 0,C 180,E1 -27381.706,E2 -27381.706} C_VEL
LIN {X 0,Y 87.653,Z 280.308,A -85,B 0,C 180,E1 -27383.017,E2 -27383.017} C_VEL
LIN {X 0,Y 89.71,Z 283.618,A -85,B 0,C 180,E1 -27385.263,E2 -27385.263} C_VEL
LIN {X 0,Y 91.64,Z 287.732,A -85,B 0,C 180,E1 -27387.559,E2 -27387.559} C_VEL
LIN {X 0,Y 96.62,Z 300.189,A -85,B 0,C 180,E1 -27393.693,E2 -27393.693} C_VEL
LIN {X 0,Y 99.805,Z 311.434,A -85,B 0,C 180,E1 -27398.687,E2 -27398.687} C_VEL
LIN {X 0,Y 100.111,Z 314.228,A -85,B 0,C 180,E1 -27399.778,E2 -27399.778} C_VEL
LIN {X 0,Y 99.538,Z 324.706,A -85,B 0,C 180,E1 -27403.635,E2 -27403.635} C_VEL
LIN {X 0,Y 98.147,Z 336.17,A -85,B 0,C 180,E1 -27408.517,E2 -27408.517} C_VEL
LIN {X 0,Y 96.8,Z 345.526,A -85,B 0,C 180,E1 -27413.345,E2 -27413.345} C_VEL
LIN {X 0,Y 93.891,Z 352.159,A -85,B 0,C 180,E1 -27417.131,E2 -27417.131} C_VEL
LIN {X 0,Y 89.969,Z 360.673,A -85,B 0,C 180,E1 -27423.307,E2 -27423.307} C_VEL
LIN {X 0,Y 86.983,Z 367.441,A -85,B 0,C 180,E1 -27429.914,E2 -27429.914} C_VEL
LIN {X 0,Y 85.098,Z 373.665,A -85,B 0,C 180,E1 -27438.082,E2 -27438.082} C_VEL
LIN {X 0,Y 84.639,Z 377.698,A -85,B 0,C 180,E1 -27445.234,E2 -27445.234} C_VEL
LIN {X 0,Y 84.689,Z 379.775,A -85,B 0,C 180,E1 -27449.997,E2 -27449.997} C_VEL
LIN {X 0,Y 84.497,Z 381.299,A -85,B 0,C 180,E1 -27454.768,E2 -27454.768} C_VEL
LIN {X 0,Y 85.164,Z 383.144,A -85,B 0,C 180,E1 -27464.331,E2 -27464.331} C_VEL
LIN {X 0,Y 88.017,Z 383.582,A -85,B 0,C 180,E1 -27473.528,E2 -27473.528} C_VEL
LIN {X 0,Y 93.209,Z 382.627,A -85,B 0,C 180,E1 -27481.854,E2 -27481.854} C_VEL
LIN {X 0,Y 100.213,Z 380.254,A -85,B 0,C 180,E1 -27489.134,E2 -27489.134} C_VEL
LIN {X 0,Y 108.638,Z 376.467,A -85,B 0,C 180,E1 -27495.363,E2 -27495.363} C_VEL
LIN {X 0,Y 115.834,Z 372.559,A -85,B 0,C 180,E1 -27499.321,E2 -27499.321} C_VEL
LIN {X 0,Y 120.974,Z 369.438,A -85,B 0,C 180,E1 -27501.651,E2 -27501.651} C_VEL
LIN {X 0,Y 125.663,Z 365.958,A -85,B 0,C 180,E1 -27504.185,E2 -27504.185} C_VEL
LIN {X 0,Y 129.693,Z 362.489,A -85,B 0,C 180,E1 -27506.696,E2 -27506.696} C_VEL
LIN {X 0,Y 130.465,Z 361.678,A -85,B 0,C 180,E1 -27507.4,E2 -27507.4} C_VEL
LIN {X 0,Y 131.827,Z 359.062,A -85,B 0,C 180,E1 -27511.322,E2 -27511.322} C_VEL
LIN {X 0,Y 132.598,Z 357.304,A -85,B 0,C 180,E1 -27514.906,E2 -27514.906} C_VEL
LIN {X 0,Y 133.243,Z 356.079,A -85,B 0,C 180,E1 -27518.327,E2 -27518.327} C_VEL
LIN {X 0,Y 133.665,Z 355.403,A -85,B 0,C 180,E1 -27521.605,E2 -27521.605} C_VEL
LIN {X 0,Y 133.663,Z 355.409,A -85,B 0,C 180,E1 -27524.753,E2 -27524.753} C_VEL
LIN {X 0,Y 133.536,Z 355.812,A -85,B 0,C 180,E1 -27527.842,E2 -27527.842} C_VEL
LIN {X 0,Y 133.073,Z 356.775,A -85,B 0,C 180,E1 -27530.879,E2 -27530.879} C_VEL
LIN {X 0,Y 132.075,Z 358.203,A -85,B 0,C 180,E1 -27533.886,E2 -27533.886} C_VEL
LIN {X 0,Y 129.969,Z 359.832,A -85,B 0,C 180,E1 -27535.158,E2 -27535.158} C_VEL
LIN {X 0,Y 122.601,Z 364.549,A -85,B 0,C 180,E1 -27538.193,E2 -27538.193} C_VEL
LIN {X 0,Y 115.691,Z 368.296,A -85,B 0,C 180,E1 -27541.587,E2 -27541.587} C_VEL
LIN {X 0,Y 109.148,Z 371.211,A -85,B 0,C 180,E1 -27545.437,E2 -27545.437} C_VEL
LIN {X 0,Y 100.438,Z 374.13,A -85,B 0,C 180,E1 -27552.111,E2 -27552.111} C_VEL
LIN {X 0,Y 95.583,Z 375.141,A -85,B 0,C 180,E1 -27557.097,E2 -27557.097} C_VEL
LIN {X 0,Y 91.389,Z 375.414,A -85,B 0,C 180,E1 -27562.665,E2 -27562.665} C_VEL
LIN {X 0,Y 88.093,Z 374.983,A -85,B 0,C 180,E1 -27568.655,E2 -27568.655} C_VEL
LIN {X 0,Y 85.73,Z 373.836,A -85,B 0,C 180,E1 -27575.009,E2 -27575.009} C_VEL
LIN {X 0,Y 83.946,Z 370.674,A -85,B 0,C 180,E1 -27584.894,E2 -27584.894} C_VEL
LIN {X 0,Y 84.376,Z 366.096,A -85,B 0,C 180,E1 -27594.338,E2 -27594.338} C_VEL
LIN {X 0,Y 85.054,Z 363.787,A -85,B 0,C 180,E1 -27597.993,E2 -27597.993} C_VEL
LIN {X 0,Y 85.299,Z 361.288,A -85,B 0,C 180,E1 -27601.583,E2 -27601.583} C_VEL
LIN {X 0,Y 84.803,Z 358.544,A -85,B 0,C 180,E1 -27605.12,E2 -27605.12} C_VEL
LIN {X 0,Y 83.95,Z 351.274,A -85,B 0,C 180,E1 -27613.193,E2 -27613.193} C_VEL
LIN {X 0,Y 85.036,Z 347.685,A -85,B 0,C 180,E1 -27616.355,E2 -27616.355} C_VEL
LIN {X 0,Y 89.007,Z 339.578,A -85,B 0,C 180,E1 -27621.981,E2 -27621.981} C_VEL
LIN {X 0,Y 93.947,Z 329.173,A -85,B 0,C 180,E1 -27627.323,E2 -27627.323} C_VEL
LIN {X 0,Y 96.109,Z 323.974,A -85,B 0,C 180,E1 -27629.479,E2 -27629.479} C_VEL
LIN {X 0,Y 95.892,Z 315.713,A -85,B 0,C 180,E1 -27633.679,E2 -27633.679} C_VEL
LIN {X 0,Y 94.463,Z 308.242,A -85,B 0,C 180,E1 -27637.651,E2 -27637.651} C_VEL
LIN {X 0,Y 93.381,Z 304.809,A -85,B 0,C 180,E1 -27639.595,E2 -27639.595} C_VEL
LIN {X 0,Y 89.499,Z 295.732,A -85,B 0,C 180,E1 -27645.36,E2 -27645.36} C_VEL
LIN {X 0,Y 87.557,Z 292.004,A -85,B 0,C 180,E1 -27647.983,E2 -27647.983} C_VEL
LIN {X 0,Y 85.237,Z 288.019,A -85,B 0,C 180,E1 -27651.109,E2 -27651.109} C_VEL
LIN {X 0,Y 83.853,Z 286.298,A -85,B 0,C 180,E1 -27652.811,E2 -27652.811} C_VEL
LIN {X 0,Y 81.983,Z 283.106,A -85,B 0,C 180,E1 -27655.619,E2 -27655.619} C_VEL
LIN {X 0,Y 79.938,Z 280.43,A -85,B 0,C 180,E1 -27658.475,E2 -27658.475} C_VEL
LIN {X 0,Y 79.425,Z 278.591,A -85,B 0,C 180,E1 -27659.708,E2 -27659.708} C_VEL
LIN {X 0,Y 79.451,Z 278.573,A -85,B 0,C 180,E1 -27668.261,E2 -27668.261} C_VEL
LIN {X 0,Y 79.489,Z 278.566,A -85,B 0,C 180,E1 -27675.021,E2 -27675.021} C_VEL
LIN {X 0,Y 79.461,Z 278.586,A -85,B 0,C 180,E1 -27682.755,E2 -27682.755} C_VEL
LIN {X 0,Y 79.482,Z 278.563,A -85,B 0,C 180,E1 -27692.161,E2 -27692.161} C_VEL
LIN {X 0,Y 79.512,Z 278.568,A -85,B 0,C 180,E1 -27699.304,E2 -27699.304} C_VEL
LIN {X 0,Y 79.826,Z 278.523,A -85,B 0,C 180,E1 -27705.582,E2 -27705.582} C_VEL
LIN {X 0,Y 79.969,Z 278.523,A -85,B 0,C 180,E1 -27709.885,E2 -27709.885} C_VEL
LIN {X 0,Y 80.647,Z 278.436,A -85,B 0,C 180,E1 -27720.008,E2 -27720.008} C_VEL
LIN {X 0,Y 79.972,Z 278.518,A -85,B 0,C 180,E1 -27730.131,E2 -27730.131} C_VEL
LIN {X 0,Y 79.757,Z 278.608,A -85,B 0,C 180,E1 -27735.501,E2 -27735.501} C_VEL
LIN {X 0,Y 80.571,Z 281.236,A -85,B 0,C 180,E1 -27737.132,E2 -27737.132} C_VEL
LIN {X 0,Y 83.063,Z 284.15,A -85,B 0,C 180,E1 -27740.274,E2 -27740.274} C_VEL
LIN {X 0,Y 85.391,Z 288.75,A -85,B 0,C 180,E1 -27743.502,E2 -27743.502} C_VEL
LIN {X 0,Y 88.74,Z 297.04,A -85,B 0,C 180,E1 -27748.38,E2 -27748.38} C_VEL
LIN {X 0,Y 91.706,Z 305.934,A -85,B 0,C 180,E1 -27753.104,E2 -27753.104} C_VEL
LIN {X 0,Y 94.007,Z 315.4,A -85,B 0,C 180,E1 -27757.732,E2 -27757.732} C_VEL
LIN {X 0,Y 93.192,Z 325.517,A -85,B 0,C 180,E1 -27761.791,E2 -27761.791} C_VEL
LIN {X 0,Y 91.712,Z 335.575,A -85,B 0,C 180,E1 -27766.392,E2 -27766.392} C_VEL
LIN {X 0,Y 90.213,Z 344.756,A -85,B 0,C 180,E1 -27771.444,E2 -27771.444} C_VEL
LIN {X 0,Y 88.843,Z 348.425,A -85,B 0,C 180,E1 -27773.606,E2 -27773.606} C_VEL
LIN {X 0,Y 85.005,Z 356.178,A -85,B 0,C 180,E1 -27778.884,E2 -27778.884} C_VEL
LIN {X 0,Y 81.347,Z 363.772,A -85,B 0,C 180,E1 -27785.769,E2 -27785.769} C_VEL
LIN {X 0,Y 78.613,Z 370.736,A -85,B 0,C 180,E1 -27794.44,E2 -27794.44} C_VEL
LIN {X 0,Y 77.651,Z 375.354,A -85,B 0,C 180,E1 -27802.194,E2 -27802.194} C_VEL
LIN {X 0,Y 77.636,Z 378.803,A -85,B 0,C 180,E1 -27809.997,E2 -27809.997} C_VEL
LIN {X 0,Y 77.454,Z 380.44,A -85,B 0,C 180,E1 -27815.203,E2 -27815.203} C_VEL
LIN {X 0,Y 78.294,Z 382.484,A -85,B 0,C 180,E1 -27825.619,E2 -27825.619} C_VEL
LIN {X 0,Y 81.533,Z 383.099,A -85,B 0,C 180,E1 -27835.527,E2 -27835.527} C_VEL
LIN {X 0,Y 87.231,Z 382.368,A -85,B 0,C 180,E1 -27844.328,E2 -27844.328} C_VEL
LIN {X 0,Y 94.789,Z 380.251,A -85,B 0,C 180,E1 -27851.855,E2 -27851.855} C_VEL
LIN {X 0,Y 103.759,Z 376.666,A -85,B 0,C 180,E1 -27858.162,E2 -27858.162} C_VEL
LIN {X 0,Y 114,Z 371.592,A -85,B 0,C 180,E1 -27863.264,E2 -27863.264} C_VEL
LIN {X 0,Y 116.709,Z 370.031,A -85,B 0,C 180,E1 -27864.381,E2 -27864.381} C_VEL
LIN {X 0,Y 121.569,Z 366.756,A -85,B 0,C 180,E1 -27866.953,E2 -27866.953} C_VEL
LIN {X 0,Y 123.897,Z 364.991,A -85,B 0,C 180,E1 -27868.303,E2 -27868.303} C_VEL
LIN {X 0,Y 124.936,Z 363.906,A -85,B 0,C 180,E1 -27869.578,E2 -27869.578} C_VEL
LIN {X 0,Y 126.178,Z 361.868,A -85,B 0,C 180,E1 -27873.533,E2 -27873.533} C_VEL
LIN {X 0,Y 126.979,Z 360.45,A -85,B 0,C 180,E1 -27877.2,E2 -27877.2} C_VEL
LIN {X 0,Y 127.61,Z 359.565,A -85,B 0,C 180,E1 -27880.699,E2 -27880.699} C_VEL
LIN {X 0,Y 127.747,Z 359.337,A -85,B 0,C 180,E1 -27884.028,E2 -27884.028} C_VEL
LIN {X 0,Y 127.61,Z 359.615,A -85,B 0,C 180,E1 -27887.268,E2 -27887.268} C_VEL
LIN {X 0,Y 127.018,Z 360.41,A -85,B 0,C 180,E1 -27890.44,E2 -27890.44} C_VEL
LIN {X 0,Y 126.408,Z 361.056,A -85,B 0,C 180,E1 -27892.005,E2 -27892.005} C_VEL
LIN {X 0,Y 123.681,Z 362.857,A -85,B 0,C 180,E1 -27893.469,E2 -27893.469} C_VEL
LIN {X 0,Y 116.189,Z 367.016,A -85,B 0,C 180,E1 -27896.526,E2 -27896.526} C_VEL
LIN {X 0,Y 105.478,Z 371.711,A -85,B 0,C 180,E1 -27901.973,E2 -27901.973} C_VEL
LIN {X 0,Y 96.274,Z 374.563,A -85,B 0,C 180,E1 -27908.388,E2 -27908.388} C_VEL
LIN {X 0,Y 90.827,Z 375.588,A -85,B 0,C 180,E1 -27913.415,E2 -27913.415} C_VEL
LIN {X 0,Y 86.135,Z 375.898,A -85,B 0,C 180,E1 -27919.04,E2 -27919.04} C_VEL
LIN {X 0,Y 82.298,Z 375.522,A -85,B 0,C 180,E1 -27925.267,E2 -27925.267} C_VEL
LIN {X 0,Y 79.379,Z 374.393,A -85,B 0,C 180,E1 -27932.078,E2 -27932.078} C_VEL
LIN {X 0,Y 77.48,Z 372.449,A -85,B 0,C 180,E1 -27939.404,E2 -27939.404} C_VEL
LIN {X 0,Y 76.819,Z 368.264,A -85,B 0,C 180,E1 -27950.181,E2 -27950.181} C_VEL
LIN {X 0,Y 78.023,Z 363.559,A -85,B 0,C 180,E1 -27958.696,E2 -27958.696} C_VEL
LIN {X 0,Y 80.389,Z 357.553,A -85,B 0,C 180,E1 -27966.836,E2 -27966.836} C_VEL
LIN {X 0,Y 83.777,Z 350.313,A -85,B 0,C 180,E1 -27974.181,E2 -27974.181} C_VEL
LIN {X 0,Y 85.036,Z 347.685,A -85,B 0,C 180,E1 -27976.355,E2 -27976.355} C_VEL
LIN {X 0,Y 86.275,Z 343.962,A -85,B 0,C 180,E1 -27979.311,E2 -27979.311} C_VEL
LIN {X 0,Y 86.928,Z 337.425,A -85,B 0,C 180,E1 -27984.23,E2 -27984.23} C_VEL
LIN {X 0,Y 87.832,Z 330.339,A -85,B 0,C 180,E1 -27988.774,E2 -27988.774} C_VEL
LIN {X 0,Y 89.37,Z 325.751,A -85,B 0,C 180,E1 -27990.993,E2 -27990.993} C_VEL
LIN {X 0,Y 89.702,Z 321.364,A -85,B 0,C 180,E1 -27993.371,E2 -27993.371} C_VEL
LIN {X 0,Y 89.342,Z 315.841,A -85,B 0,C 180,E1 -27996.478,E2 -27996.478} C_VEL
LIN {X 0,Y 88.129,Z 309.694,A -85,B 0,C 180,E1 -28000.173,E2 -28000.173} C_VEL
LIN {X 0,Y 84.436,Z 300.172,A -85,B 0,C 180,E1 -28006.81,E2 -28006.81} C_VEL
LIN {X 0,Y 80.701,Z 292.999,A -85,B 0,C 180,E1 -28012.852,E2 -28012.852} C_VEL
LIN {X 0,Y 78.459,Z 289.117,A -85,B 0,C 180,E1 -28016.611,E2 -28016.611} C_VEL
LIN {X 0,Y 76.661,Z 286.81,A -85,B 0,C 180,E1 -28019.448,E2 -28019.448} C_VEL
LIN {X 0,Y 75.907,Z 285.073,A -85,B 0,C 180,E1 -28021.099,E2 -28021.099} C_VEL
LIN {X 0,Y 73.204,Z 282.033,A -85,B 0,C 180,E1 -28026.073,E2 -28026.073} C_VEL
LIN {X 0,Y 72.385,Z 279.454,A -85,B 0,C 180,E1 -28028.706,E2 -28028.706} C_VEL
LIN {X 0,Y 72.326,Z 279.448,A -85,B 0,C 180,E1 -28037.155,E2 -28037.155} C_VEL
LIN {X 0,Y 72.344,Z 279.472,A -85,B 0,C 180,E1 -28044.359,E2 -28044.359} C_VEL
LIN {X 0,Y 72.39,Z 279.439,A -85,B 0,C 180,E1 -28050.971,E2 -28050.971} C_VEL
LIN {X 0,Y 72.393,Z 279.466,A -85,B 0,C 180,E1 -28057.16,E2 -28057.16} C_VEL
LIN {X 0,Y 72.722,Z 279.403,A -85,B 0,C 180,E1 -28065.119,E2 -28065.119} C_VEL
LIN {X 0,Y 72.86,Z 279.409,A -85,B 0,C 180,E1 -28068.886,E2 -28068.886} C_VEL
LIN {X 0,Y 73.573,Z 279.317,A -85,B 0,C 180,E1 -28080.009,E2 -28080.009} C_VEL
LIN {X 0,Y 72.974,Z 279.559,A -85,B 0,C 180,E1 -28087.271,E2 -28087.271} C_VEL
LIN {X 0,Y 73.778,Z 281.986,A -85,B 0,C 180,E1 -28089.432,E2 -28089.432} C_VEL
LIN {X 0,Y 75.758,Z 284.325,A -85,B 0,C 180,E1 -28092.867,E2 -28092.867} C_VEL
LIN {X 0,Y 76.351,Z 285.183,A -85,B 0,C 180,E1 -28093.891,E2 -28093.891} C_VEL
LIN {X 0,Y 77.994,Z 288.283,A -85,B 0,C 180,E1 -28096.825,E2 -28096.825} C_VEL
LIN {X 0,Y 79.353,Z 290.113,A -85,B 0,C 180,E1 -28098.841,E2 -28098.841} C_VEL
LIN {X 0,Y 81.023,Z 293.824,A -85,B 0,C 180,E1 -28101.724,E2 -28101.724} C_VEL
LIN {X 0,Y 83.738,Z 301.281,A -85,B 0,C 180,E1 -28106.578,E2 -28106.578} C_VEL
LIN {X 0,Y 86.059,Z 309.24,A -85,B 0,C 180,E1 -28111.316,E2 -28111.316} C_VEL
LIN {X 0,Y 87.741,Z 316.864,A -85,B 0,C 180,E1 -28115.51,E2 -28115.51} C_VEL
LIN {X 0,Y 87.547,Z 321.254,A -85,B 0,C 180,E1 -28117.472,E2 -28117.472} C_VEL
LIN {X 0,Y 86.172,Z 330.869,A -85,B 0,C 180,E1 -28121.875,E2 -28121.875} C_VEL
LIN {X 0,Y 84.352,Z 341.015,A -85,B 0,C 180,E1 -28127.39,E2 -28127.39} C_VEL
LIN {X 0,Y 83.125,Z 346.241,A -85,B 0,C 180,E1 -28130.699,E2 -28130.699} C_VEL
LIN {X 0,Y 78.998,Z 354.244,A -85,B 0,C 180,E1 -28136.215,E2 -28136.215} C_VEL
LIN {X 0,Y 74.962,Z 362.123,A -85,B 0,C 180,E1 -28143.552,E2 -28143.552} C_VEL
LIN {X 0,Y 72.501,Z 367.461,A -85,B 0,C 180,E1 -28150.164,E2 -28150.164} C_VEL
LIN {X 0,Y 70.903,Z 372.685,A -85,B 0,C 180,E1 -28158.563,E2 -28158.563} C_VEL
LIN {X 0,Y 70.529,Z 376.649,A -85,B 0,C 180,E1 -28167.017,E2 -28167.017} C_VEL
LIN {X 0,Y 70.586,Z 377.786,A -85,B 0,C 180,E1 -28169.997,E2 -28169.997} C_VEL
LIN {X 0,Y 70.442,Z 379.517,A -85,B 0,C 180,E1 -28175.723,E2 -28175.723} C_VEL
LIN {X 0,Y 71.478,Z 381.781,A -85,B 0,C 180,E1 -28187.153,E2 -28187.153} C_VEL
LIN {X 0,Y 75.165,Z 382.613,A -85,B 0,C 180,E1 -28197.869,E2 -28197.869} C_VEL
LIN {X 0,Y 81.442,Z 382.074,A -85,B 0,C 180,E1 -28207.158,E2 -28207.158} C_VEL
LIN {X 0,Y 89.595,Z 380.181,A -85,B 0,C 180,E1 -28214.905,E2 -28214.905} C_VEL
LIN {X 0,Y 99.164,Z 376.908,A -85,B 0,C 180,E1 -28221.22,E2 -28221.22} C_VEL
LIN {X 0,Y 107.151,Z 373.441,A -85,B 0,C 180,E1 -28225.068,E2 -28225.068} C_VEL
LIN {X 0,Y 112.707,Z 370.628,A -85,B 0,C 180,E1 -28227.328,E2 -28227.328} C_VEL
LIN {X 0,Y 117.664,Z 367.586,A -85,B 0,C 180,E1 -28229.856,E2 -28229.856} C_VEL
LIN {X 0,Y 119.29,Z 366.106,A -85,B 0,C 180,E1 -28232.091,E2 -28232.091} C_VEL
LIN {X 0,Y 120.405,Z 364.566,A -85,B 0,C 180,E1 -28235.878,E2 -28235.878} C_VEL
LIN {X 0,Y 121.321,Z 363.444,A -85,B 0,C 180,E1 -28239.655,E2 -28239.655} C_VEL
LIN {X 0,Y 121.564,Z 363.027,A -85,B 0,C 180,E1 -28243.192,E2 -28243.192} C_VEL
LIN {X 0,Y 121.492,Z 363.143,A -85,B 0,C 180,E1 -28246.616,E2 -28246.616} C_VEL
LIN {X 0,Y 120.822,Z 363.743,A -85,B 0,C 180,E1 -28249.945,E2 -28249.945} C_VEL
LIN {X 0,Y 117.962,Z 365.395,A -85,B 0,C 180,E1 -28251.428,E2 -28251.428} C_VEL
LIN {X 0,Y 110.083,Z 369.187,A -85,B 0,C 180,E1 -28254.537,E2 -28254.537} C_VEL
LIN {X 0,Y 102.59,Z 372.109,A -85,B 0,C 180,E1 -28258.095,E2 -28258.095} C_VEL
LIN {X 0,Y 92.542,Z 375.007,A -85,B 0,C 180,E1 -28264.348,E2 -28264.348} C_VEL
LIN {X 0,Y 85.671,Z 376.16,A -85,B 0,C 180,E1 -28270.143,E2 -28270.143} C_VEL
LIN {X 0,Y 80.428,Z 376.379,A -85,B 0,C 180,E1 -28276.023,E2 -28276.023} C_VEL
LIN {X 0,Y 76.126,Z 375.898,A -85,B 0,C 180,E1 -28282.609,E2 -28282.609} C_VEL
LIN {X 0,Y 72.873,Z 374.729,A -85,B 0,C 180,E1 -28289.783,E2 -28289.783} C_VEL
LIN {X 0,Y 70.056,Z 371.607,A -85,B 0,C 180,E1 -28301.211,E2 -28301.211} C_VEL
LIN {X 0,Y 69.941,Z 366.888,A -85,B 0,C 180,E1 -28312.926,E2 -28312.926} C_VEL
LIN {X 0,Y 71.609,Z 361.774,A -85,B 0,C 180,E1 -28322.021,E2 -28322.021} C_VEL
LIN {X 0,Y 74.506,Z 355.286,A -85,B 0,C 180,E1 -28330.58,E2 -28330.58} C_VEL
LIN {X 0,Y 78.447,Z 347.506,A -85,B 0,C 180,E1 -28338.181,E2 -28338.181} C_VEL
LIN {X 0,Y 83.031,Z 338.634,A -85,B 0,C 180,E1 -28344.538,E2 -28344.538} C_VEL
LIN {X 0,Y 88.305,Z 328.065,A -85,B 0,C 180,E1 -28350.003,E2 -28350.003} C_VEL
LIN {X 0,Y 89.37,Z 325.751,A -85,B 0,C 180,E1 -28350.993,E2 -28350.993} C_VEL
LIN {X 0,Y 89.996,Z 322.84,A -85,B 0,C 180,E1 -28352.43,E2 -28352.43} C_VEL
LIN {X 0,Y 89.551,Z 320.091,A -85,B 0,C 180,E1 -28354.127,E2 -28354.127} C_VEL
LIN {X 0,Y 87.633,Z 316.54,A -85,B 0,C 180,E1 -28356.957,E2 -28356.957} C_VEL
LIN {X 0,Y 81.228,Z 308.946,A -85,B 0,C 180,E1 -28364.681,E2 -28364.681} C_VEL
LIN {X 0,Y 79.953,Z 306.304,A -85,B 0,C 180,E1 -28366.958,E2 -28366.958} C_VEL
LIN {X 0,Y 77.872,Z 301.513,A -85,B 0,C 180,E1 -28371.165,E2 -28371.165} C_VEL
LIN {X 0,Y 74.374,Z 294.606,A -85,B 0,C 180,E1 -28378.198,E2 -28378.198} C_VEL
LIN {X 0,Y 72.118,Z 290.675,A -85,B 0,C 180,E1 -28383.101,E2 -28383.101} C_VEL
LIN {X 0,Y 70.311,Z 288.616,A -85,B 0,C 180,E1 -28386.921,E2 -28386.921} C_VEL
LIN {X 0,Y 69.287,Z 285.863,A -85,B 0,C 180,E1 -28390.321,E2 -28390.321} C_VEL
LIN {X 0,Y 66.461,Z 283.461,A -85,B 0,C 180,E1 -28398.39,E2 -28398.39} C_VEL
LIN {X 0,Y 65.225,Z 280.347,A -85,B 0,C 180,E1 -28406.029,E2 -28406.029} C_VEL
LIN {X 0,Y 65.245,Z 280.351,A -85,B 0,C 180,E1 -28414.489,E2 -28414.489} C_VEL
LIN {X 0,Y 65.626,Z 280.282,A -85,B 0,C 180,E1 -28424.554,E2 -28424.554} C_VEL
LIN {X 0,Y 65.84,Z 280.42,A -85,B 0,C 180,E1 -28431.571,E2 -28431.571} C_VEL
LIN {X 0,Y 67.293,Z 283.118,A -85,B 0,C 180,E1 -28438.14,E2 -28438.14} C_VEL
LIN {X 0,Y 69.937,Z 285.892,A -85,B 0,C 180,E1 -28445.235,E2 -28445.235} C_VEL
LIN {X 0,Y 71.057,Z 288.589,A -85,B 0,C 180,E1 -28448.462,E2 -28448.462} C_VEL
LIN {X 0,Y 72.388,Z 290.274,A -85,B 0,C 180,E1 -28451.206,E2 -28451.206} C_VEL
LIN {X 0,Y 73.81,Z 293.247,A -85,B 0,C 180,E1 -28454.379,E2 -28454.379} C_VEL
LIN {X 0,Y 74.979,Z 294.783,A -85,B 0,C 180,E1 -28456.341,E2 -28456.341} C_VEL
LIN {X 0,Y 76.475,Z 298.408,A -85,B 0,C 180,E1 -28459.578,E2 -28459.578} C_VEL
LIN {X 0,Y 78.791,Z 306.027,A -85,B 0,C 180,E1 -28465.077,E2 -28465.077} C_VEL
LIN {X 0,Y 80.643,Z 313.436,A -85,B 0,C 180,E1 -28469.94,E2 -28469.94} C_VEL
LIN {X 0,Y 81.727,Z 320.045,A -85,B 0,C 180,E1 -28473.993,E2 -28473.993} C_VEL
LIN {X 0,Y 80.439,Z 328.577,A -85,B 0,C 180,E1 -28478.151,E2 -28478.151} C_VEL
LIN {X 0,Y 78.218,Z 339.059,A -85,B 0,C 180,E1 -28484.04,E2 -28484.04} C_VEL
LIN {X 0,Y 76.559,Z 346.034,A -85,B 0,C 180,E1 -28488.739,E2 -28488.739} C_VEL
LIN {X 0,Y 71.566,Z 355.09,A -85,B 0,C 180,E1 -28495.617,E2 -28495.617} C_VEL
LIN {X 0,Y 67.419,Z 362.706,A -85,B 0,C 180,E1 -28503.699,E2 -28503.699} C_VEL
LIN {X 0,Y 64.429,Z 369.678,A -85,B 0,C 180,E1 -28514.171,E2 -28514.171} C_VEL
LIN {X 0,Y 63.529,Z 374.782,A -85,B 0,C 180,E1 -28524.755,E2 -28524.755} C_VEL
LIN {X 0,Y 63.548,Z 376.743,A -85,B 0,C 180,E1 -28529.997,E2 -28529.997} C_VEL
LIN {X 0,Y 63.408,Z 378.591,A -85,B 0,C 180,E1 -28536.36,E2 -28536.36} C_VEL
LIN {X 0,Y 64.73,Z 381.012,A -85,B 0,C 180,E1 -28549.006,E2 -28549.006} C_VEL
LIN {X 0,Y 68.95,Z 382.061,A -85,B 0,C 180,E1 -28560.636,E2 -28560.636} C_VEL
LIN {X 0,Y 75.884,Z 381.78,A -85,B 0,C 180,E1 -28570.41,E2 -28570.41} C_VEL
LIN {X 0,Y 85.165,Z 379.983,A -85,B 0,C 180,E1 -28578.677,E2 -28578.677} C_VEL
LIN {X 0,Y 94.875,Z 377.064,A -85,B 0,C 180,E1 -28584.568,E2 -28584.568} C_VEL
LIN {X 0,Y 106.143,Z 372.573,A -85,B 0,C 180,E1 -28589.398,E2 -28589.398} C_VEL
LIN {X 0,Y 109.01,Z 371.186,A -85,B 0,C 180,E1 -28590.496,E2 -28590.496} C_VEL
LIN {X 0,Y 111.682,Z 369.772,A -85,B 0,C 180,E1 -28591.758,E2 -28591.758} C_VEL
LIN {X 0,Y 113.376,Z 368.415,A -85,B 0,C 180,E1 -28594.277,E2 -28594.277} C_VEL
LIN {X 0,Y 114.635,Z 367.111,A -85,B 0,C 180,E1 -28598.411,E2 -28598.411} C_VEL
LIN {X 0,Y 115.18,Z 366.449,A -85,B 0,C 180,E1 -28602.231,E2 -28602.231} C_VEL
LIN {X 0,Y 115.169,Z 366.363,A -85,B 0,C 180,E1 -28605.866,E2 -28605.866} C_VEL
LIN {X 0,Y 114.862,Z 366.541,A -85,B 0,C 180,E1 -28607.628,E2 -28607.628} C_VEL
LIN {X 0,Y 112.349,Z 367.773,A -85,B 0,C 180,E1 -28609.178,E2 -28609.178} C_VEL
LIN {X 0,Y 104.274,Z 371.104,A -85,B 0,C 180,E1 -28612.247,E2 -28612.247} C_VEL
LIN {X 0,Y 96.54,Z 373.667,A -85,B 0,C 180,E1 -28615.818,E2 -28615.818} C_VEL
LIN {X 0,Y 89.318,Z 375.471,A -85,B 0,C 180,E1 -28619.992,E2 -28619.992} C_VEL
LIN {X 0,Y 82.678,Z 376.512,A -85,B 0,C 180,E1 -28624.868,E2 -28624.868} C_VEL
LIN {X 0,Y 76.728,Z 376.873,A -85,B 0,C 180,E1 -28630.547,E2 -28630.547} C_VEL
LIN {X 0,Y 71.622,Z 376.558,A -85,B 0,C 180,E1 -28637.11,E2 -28637.11} C_VEL
LIN {X 0,Y 67.516,Z 375.482,A -85,B 0,C 180,E1 -28644.594,E2 -28644.594} C_VEL
LIN {X 0,Y 64.504,Z 373.654,A -85,B 0,C 180,E1 -28652.996,E2 -28652.996} C_VEL
LIN {X 0,Y 62.824,Z 370.988,A -85,B 0,C 180,E1 -28662.145,E2 -28662.145} C_VEL
LIN {X 0,Y 62.962,Z 366.323,A -85,B 0,C 180,E1 -28673.975,E2 -28673.975} C_VEL
LIN {X 0,Y 64.967,Z 360.731,A -85,B 0,C 180,E1 -28684.364,E2 -28684.364} C_VEL
LIN {X 0,Y 68.318,Z 353.97,A -85,B 0,C 180,E1 -28693.57,E2 -28693.57} C_VEL
LIN {X 0,Y 72.82,Z 345.71,A -85,B 0,C 180,E1 -28701.679,E2 -28701.679} C_VEL
LIN {X 0,Y 77.361,Z 337.402,A -85,B 0,C 180,E1 -28707.634,E2 -28707.634} C_VEL
LIN {X 0,Y 82.847,Z 326.952,A -85,B 0,C 180,E1 -28713.042,E2 -28713.042} C_VEL
LIN {X 0,Y 83.272,Z 325.72,A -85,B 0,C 180,E1 -28713.632,E2 -28713.632} C_VEL
LIN {X 0,Y 83.398,Z 319.821,A -85,B 0,C 180,E1 -28717.249,E2 -28717.249} C_VEL
LIN {X 0,Y 82.618,Z 314.328,A -85,B 0,C 180,E1 -28720.86,E2 -28720.86} C_VEL
LIN {X 0,Y 79.953,Z 306.304,A -85,B 0,C 180,E1 -28726.958,E2 -28726.958} C_VEL
LIN {X 0,Y 78.811,Z 303.997,A -85,B 0,C 180,E1 -28729.089,E2 -28729.089} C_VEL
LIN {X 0,Y 76.384,Z 301.438,A -85,B 0,C 180,E1 -28732.594,E2 -28732.594} C_VEL
LIN {X 0,Y 71.679,Z 298.594,A -85,B 0,C 180,E1 -28739.133,E2 -28739.133} C_VEL
LIN {X 0,Y 67.672,Z 295.606,A -85,B 0,C 180,E1 -28746.487,E2 -28746.487} C_VEL
LIN {X 0,Y 67.103,Z 294.785,A -85,B 0,C 180,E1 -28748.003,E2 -28748.003} C_VEL
LIN {X 0,Y 66.106,Z 292.143,A -85,B 0,C 180,E1 -28751.926,E2 -28751.926} C_VEL
LIN {X 0,Y 63.744,Z 289.597,A -85,B 0,C 180,E1 -28760.518,E2 -28760.518} C_VEL
LIN {X 0,Y 63.084,Z 287.353,A -85,B 0,C 180,E1 -28766.163,E2 -28766.163} C_VEL
LIN {X 0,Y 62.32,Z 286.821,A -85,B 0,C 180,E1 -28774.454,E2 -28774.454} C_VEL
LIN {X 0,Y 63.077,Z 286.874,A -85,B 0,C 180,E1 -28787.135,E2 -28787.135} C_VEL
LIN {X 0,Y 63.863,Z 287.911,A -85,B 0,C 180,E1 -28792.093,E2 -28792.093} C_VEL
LIN {X 0,Y 66.704,Z 291.878,A -85,B 0,C 180,E1 -28803.03,E2 -28803.03} C_VEL
LIN {X 0,Y 69.18,Z 296.997,A -85,B 0,C 180,E1 -28810.549,E2 -28810.549} C_VEL
LIN {X 0,Y 71.476,Z 301.458,A -85,B 0,C 180,E1 -28816.009,E2 -28816.009} C_VEL
LIN {X 0,Y 73.198,Z 308.093,A -85,B 0,C 180,E1 -28821.54,E2 -28821.54} C_VEL
LIN {X 0,Y 74.972,Z 316.738,A -85,B 0,C 180,E1 -28827.96,E2 -28827.96} C_VEL
LIN {X 0,Y 75.685,Z 321.831,A -85,B 0,C 180,E1 -28831.469,E2 -28831.469} C_VEL
LIN {X 0,Y 74.245,Z 329.758,A -85,B 0,C 180,E1 -28835.747,E2 -28835.747} C_VEL
LIN {X 0,Y 71.763,Z 339.669,A -85,B 0,C 180,E1 -28841.861,E2 -28841.861} C_VEL
LIN {X 0,Y 70.401,Z 344.846,A -85,B 0,C 180,E1 -28845.666,E2 -28845.666} C_VEL
LIN {X 0,Y 68.626,Z 348.393,A -85,B 0,C 180,E1 -28848.263,E2 -28848.263} C_VEL
LIN {X 0,Y 63.363,Z 357.219,A -85,B 0,C 180,E1 -28856.314,E2 -28856.314} C_VEL
LIN {X 0,Y 59.37,Z 364.313,A -85,B 0,C 180,E1 -28865.52,E2 -28865.52} C_VEL
LIN {X 0,Y 57.086,Z 369.991,A -85,B 0,C 180,E1 -28875.742,E2 -28875.742} C_VEL
LIN {X 0,Y 56.498,Z 373.678,A -85,B 0,C 180,E1 -28884.466,E2 -28884.466} C_VEL
LIN {X 0,Y 56.52,Z 375.599,A -85,B 0,C 180,E1 -28889.996,E2 -28889.996} C_VEL
LIN {X 0,Y 56.409,Z 377.556,A -85,B 0,C 180,E1 -28897.153,E2 -28897.153} C_VEL
LIN {X 0,Y 58.071,Z 380.24,A -85,B 0,C 180,E1 -28911.285,E2 -28911.285} C_VEL
LIN {X 0,Y 62.931,Z 381.475,A -85,B 0,C 180,E1 -28923.94,E2 -28923.94} C_VEL
LIN {X 0,Y 70.61,Z 381.405,A -85,B 0,C 180,E1 -28934.16,E2 -28934.16} C_VEL
LIN {X 0,Y 80.113,Z 380.008,A -85,B 0,C 180,E1 -28942.137,E2 -28942.137} C_VEL
LIN {X 0,Y 90.936,Z 377.232,A -85,B 0,C 180,E1 -28948.222,E2 -28948.222} C_VEL
LIN {X 0,Y 102.717,Z 373.004,A -85,B 0,C 180,E1 -28952.801,E2 -28952.801} C_VEL
LIN {X 0,Y 105.652,Z 371.737,A -85,B 0,C 180,E1 -28953.894,E2 -28953.894} C_VEL
LIN {X 0,Y 107.529,Z 370.462,A -85,B 0,C 180,E1 -28956.905,E2 -28956.905} C_VEL
LIN {X 0,Y 108.467,Z 369.582,A -85,B 0,C 180,E1 -28961.091,E2 -28961.091} C_VEL
LIN {X 0,Y 108.634,Z 369.275,A -85,B 0,C 180,E1 -28965.954,E2 -28965.954} C_VEL
LIN {X 0,Y 106.904,Z 369.98,A -85,B 0,C 180,E1 -28966.691,E2 -28966.691} C_VEL
LIN {X 0,Y 100.206,Z 372.412,A -85,B 0,C 180,E1 -28969.067,E2 -28969.067} C_VEL
LIN {X 0,Y 92.149,Z 374.724,A -85,B 0,C 180,E1 -28972.495,E2 -28972.495} C_VEL
LIN {X 0,Y 84.479,Z 376.3,A -85,B 0,C 180,E1 -28976.618,E2 -28976.618} C_VEL
LIN {X 0,Y 77.333,Z 377.185,A -85,B 0,C 180,E1 -28981.576,E2 -28981.576} C_VEL
LIN {X 0,Y 70.873,Z 377.35,A -85,B 0,C 180,E1 -28987.446,E2 -28987.446} C_VEL
LIN {X 0,Y 65.3,Z 376.794,A -85,B 0,C 180,E1 -28994.403,E2 -28994.403} C_VEL
LIN {X 0,Y 60.829,Z 375.558,A -85,B 0,C 180,E1 -29002.447,E2 -29002.447} C_VEL
LIN {X 0,Y 57.617,Z 373.61,A -85,B 0,C 180,E1 -29011.376,E2 -29011.376} C_VEL
LIN {X 0,Y 55.517,Z 369.499,A -85,B 0,C 180,E1 -29025.428,E2 -29025.428} C_VEL
LIN {X 0,Y 56.355,Z 364.49,A -85,B 0,C 180,E1 -29038.003,E2 -29038.003} C_VEL
LIN {X 0,Y 59.048,Z 358.428,A -85,B 0,C 180,E1 -29049.084,E2 -29049.084} C_VEL
LIN {X 0,Y 63.249,Z 350.879,A -85,B 0,C 180,E1 -29058.969,E2 -29058.969} C_VEL
LIN {X 0,Y 68.334,Z 342.284,A -85,B 0,C 180,E1 -29066.866,E2 -29066.866} C_VEL
LIN {X 0,Y 74.193,Z 332.138,A -85,B 0,C 180,E1 -29073.397,E2 -29073.397} C_VEL
LIN {X 0,Y 76.953,Z 327.002,A -85,B 0,C 180,E1 -29075.9,E2 -29075.9} C_VEL
LIN {X 0,Y 77.222,Z 322.126,A -85,B 0,C 180,E1 -29079.167,E2 -29079.167} C_VEL
LIN {X 0,Y 76.439,Z 316.264,A -85,B 0,C 180,E1 -29083.553,E2 -29083.553} C_VEL
LIN {X 0,Y 74.449,Z 309.757,A -85,B 0,C 180,E1 -29089.294,E2 -29089.294} C_VEL
LIN {X 0,Y 72.019,Z 303.949,A -85,B 0,C 180,E1 -29095.188,E2 -29095.188} C_VEL
LIN {X 0,Y 70.105,Z 299.808,A -85,B 0,C 180,E1 -29100.086,E2 -29100.086} C_VEL
LIN {X 0,Y 68.4,Z 296.464,A -85,B 0,C 180,E1 -29104.734,E2 -29104.734} C_VEL
LIN {X 0,Y 67.103,Z 294.785,A -85,B 0,C 180,E1 -29108.003,E2 -29108.003} C_VEL
LIN {X 0,Y 66.007,Z 293.449,A -85,B 0,C 180,E1 -29111.045,E2 -29111.045} C_VEL
LIN {X 0,Y 64.217,Z 292.537,A -85,B 0,C 180,E1 -29115.954,E2 -29115.954} C_VEL
LIN {X 0,Y 61.476,Z 292.826,A -85,B 0,C 180,E1 -29124.798,E2 -29124.798} C_VEL
LIN {X 0,Y 59.933,Z 293.549,A -85,B 0,C 180,E1 -29136.323,E2 -29136.323} C_VEL
LIN {X 0,Y 60.721,Z 293.592,A -85,B 0,C 180,E1 -29146.627,E2 -29146.627} C_VEL
LIN {X 0,Y 62.258,Z 296.342,A -85,B 0,C 180,E1 -29156.775,E2 -29156.775} C_VEL
LIN {X 0,Y 63.26,Z 297.691,A -85,B 0,C 180,E1 -29160.646,E2 -29160.646} C_VEL
LIN {X 0,Y 65.496,Z 303.01,A -85,B 0,C 180,E1 -29169.273,E2 -29169.273} C_VEL
LIN {X 0,Y 66.967,Z 306.174,A -85,B 0,C 180,E1 -29173.669,E2 -29173.669} C_VEL
LIN {X 0,Y 68.243,Z 312.778,A -85,B 0,C 180,E1 -29179.721,E2 -29179.721} C_VEL
LIN {X 0,Y 69.277,Z 319.733,A -85,B 0,C 180,E1 -29185.551,E2 -29185.551} C_VEL
LIN {X 0,Y 69.597,Z 324.916,A -85,B 0,C 180,E1 -29189.501,E2 -29189.501} C_VEL
LIN {X 0,Y 66.906,Z 335.185,A -85,B 0,C 180,E1 -29195.756,E2 -29195.756} C_VEL
LIN {X 0,Y 64.24,Z 344.068,A -85,B 0,C 180,E1 -29202.395,E2 -29202.395} C_VEL
LIN {X 0,Y 63.48,Z 345.97,A -85,B 0,C 180,E1 -29203.971,E2 -29203.971} C_VEL
LIN {X 0,Y 58.487,Z 353.798,A -85,B 0,C 180,E1 -29210.882,E2 -29210.882} C_VEL
LIN {X 0,Y 53.651,Z 361.467,A -85,B 0,C 180,E1 -29220.574,E2 -29220.574} C_VEL
LIN {X 0,Y 50.974,Z 366.67,A -85,B 0,C 180,E1 -29229.833,E2 -29229.833} C_VEL
LIN {X 0,Y 49.471,Z 372.535,A -85,B 0,C 180,E1 -29244.082,E2 -29244.082} C_VEL
LIN {X 0,Y 49.492,Z 374.435,A -85,B 0,C 180,E1 -29249.996,E2 -29249.996} C_VEL
LIN {X 0,Y 49.433,Z 376.495,A -85,B 0,C 180,E1 -29258.169,E2 -29258.169} C_VEL
LIN {X 0,Y 51.533,Z 379.372,A -85,B 0,C 180,E1 -29274.146,E2 -29274.146} C_VEL
LIN {X 0,Y 57.167,Z 380.868,A -85,B 0,C 180,E1 -29287.924,E2 -29287.924} C_VEL
LIN {X 0,Y 65.69,Z 381.02,A -85,B 0,C 180,E1 -29298.491,E2 -29298.491} C_VEL
LIN {X 0,Y 75.958,Z 379.846,A -85,B 0,C 180,E1 -29306.373,E2 -29306.373} C_VEL
LIN {X 0,Y 87.408,Z 377.351,A -85,B 0,C 180,E1 -29312.178,E2 -29312.178} C_VEL
LIN {X 0,Y 99.672,Z 373.442,A -85,B 0,C 180,E1 -29316.435,E2 -29316.435} C_VEL
